H4_1_4_03_FEIL_PR2 5105.05 BOOL  ; HOVEDTAVLE 4.1_SEKSJON_SKUFF        UTLOEST MOTORV. ELLER SIKRING
H4_1_4_03_OK 1604.08 BOOL  ; HOVEDTAVLE 4.1_SEKSJON_SKUFF       DRIFT OG OK
H4_1_4_03_OK_PR2 5105.04 BOOL  ; HOVEDTAVLE 4.1_SEKSJON_SKUFF       DRIFT OG OK
H4_1_4_04_AUTO 1604.09 BOOL  ; HOVEDTAVLE 4.1_SEKSJON_SKUFF        DRIFTSIGN. FRA  NODE1_4
H4_1_4_04_AUTO_PR2 5003.03 BOOL  ; HOVEDTAVLE 4.1_SEKSJON_SKUFF        DRIFTSIGN. FRA  NODE1_4
H4_1_4_04_FEIL 1604.10 BOOL  ; HOVEDTAVLE 4.1_SEKSJON_SKUFF        UTLOEST MOTORV. ELLER SIKRING
H4_1_4_04_FEIL_PR2 5105.07 BOOL  ; HOVEDTAVLE 4.1_SEKSJON_SKUFF        UTLOEST MOTORV. ELLER SIKRING
H4_1_4_04_OK 1604.11 BOOL  ; HOVEDTAVLE 4.1_SEKSJON_SKUFF       DRIFT OG OK
H4_1_4_04_OK_PR2 5105.06 BOOL  ; HOVEDTAVLE 4.1_SEKSJON_SKUFF       DRIFT OG OK
H4_1_4_05_AUTO 1604.12 BOOL  ; HOVEDTAVLE 4.1_SEKSJON_SKUFF        DRIFTSIGN. FRA  NODE1_4
H4_1_4_05_AUTO_PR2 5003.04 BOOL  ; HOVEDTAVLE 4.1_SEKSJON_SKUFF        DRIFTSIGN. FRA  NODE1_4
H4_1_4_05_FEIL 1604.13 BOOL  ; HOVEDTAVLE 4.1_SEKSJON_SKUFF        UTLOEST MOTORV. ELLER SIKRING
H4_1_4_05_FEIL_PR2 5106.01 BOOL  ; HOVEDTAVLE 4.1_SEKSJON_SKUFF        UTLOEST MOTORV. ELLER SIKRING
H4_1_4_05_OK 1604.14 BOOL  ; HOVEDTAVLE 4.1_SEKSJON_SKUFF       DRIFT OG OK
H4_1_4_05_OK_PR2 5106.00 BOOL  ; HOVEDTAVLE 4.1_SEKSJON_SKUFF       DRIFT OG OK
H4_1_4_06_AUTO 1605.00 BOOL  ; HOVEDTAVLE 4.1_SEKSJON_SKUFF        DRIFTSIGN. FRA  NODE1_4
H4_1_4_06_AUTO_PR2 5003.05 BOOL  ; HOVEDTAVLE 4.1_SEKSJON_SKUFF        DRIFTSIGN. FRA  NODE1_4
H4_1_4_06_FEIL 1605.01 BOOL  ; HOVEDTAVLE 4.1_SEKSJON_SKUFF        UTLOEST MOTORV. ELLER SIKRING
H4_1_4_06_FEIL_PR2 5106.03 BOOL  ; HOVEDTAVLE 4.1_SEKSJON_SKUFF        UTLOEST MOTORV. ELLER SIKRING
H4_1_4_06_OK 1605.02 BOOL  ; HOVEDTAVLE 4.1_SEKSJON_SKUFF       DRIFT OG OK
H4_1_4_06_OK_PR2 5106.02 BOOL  ; HOVEDTAVLE 4.1_SEKSJON_SKUFF       DRIFT OG OK
H4_1_4_07_AUTO 1605.03 BOOL  ; HOVEDTAVLE 4.1_SEKSJON_SKUFF        DRIFTSIGN. FRA  NODE1_4
H4_1_4_07_AUTO_PR2 5003.06 BOOL  ; HOVEDTAVLE 4.1_SEKSJON_SKUFF        DRIFTSIGN. FRA  NODE1_4
H4_1_4_07_FEIL 1605.04 BOOL  ; HOVEDTAVLE 4.1_SEKSJON_SKUFF        UTLOEST MOTORV. ELLER SIKRING
H4_1_4_07_FEIL_PR2 5106.05 BOOL  ; HOVEDTAVLE 4.1_SEKSJON_SKUFF        UTLOEST MOTORV. ELLER SIKRING
H4_1_4_07_OK 1605.05 BOOL  ; HOVEDTAVLE 4.1_SEKSJON_SKUFF       DRIFT OG OK
H4_1_4_07_OK_PR2 5106.04 BOOL  ; HOVEDTAVLE 4.1_SEKSJON_SKUFF       DRIFT OG OK
H4_1_4_08_AUTO 1605.06 BOOL  ; HOVEDTAVLE 4.1_SEKSJON_SKUFF        DRIFTSIGN. FRA  NODE1_4
H4_1_4_08_AUTO_PR2 5003.07 BOOL  ; HOVEDTAVLE 4.1_SEKSJON_SKUFF        DRIFTSIGN. FRA  NODE1_4
H4_1_4_08_FEIL 1605.07 BOOL  ; HOVEDTAVLE 4.1_SEKSJON_SKUFF        UTLOEST MOTORV. ELLER SIKRING
H4_1_4_08_FEIL_PR2 5106.07 BOOL  ; HOVEDTAVLE 4.1_SEKSJON_SKUFF        UTLOEST MOTORV. ELLER SIKRING
H4_1_4_08_OK 1605.08 BOOL  ; HOVEDTAVLE 4.1_SEKSJON_SKUFF       DRIFT OG OK
H4_1_4_08_OK_PR2 5106.06 BOOL  ; HOVEDTAVLE 4.1_SEKSJON_SKUFF       DRIFT OG OK
H4_1_4_09_AUTO 1605.09 BOOL  ; HOVEDTAVLE 4.1_SEKSJON_SKUFF        DRIFTSIGN. FRA  NODE1_4
H4_1_4_09_AUTO_PR2 5004.00 BOOL  ; HOVEDTAVLE 4.1_SEKSJON_SKUFF        DRIFTSIGN. FRA  NODE1_4
H4_1_4_09_FEIL 1605.10 BOOL  ; HOVEDTAVLE 4.1_SEKSJON_SKUFF        UTLOEST MOTORV. ELLER SIKRING
H4_1_4_09_FEIL_PR2 5107.01 BOOL  ; HOVEDTAVLE 4.1_SEKSJON_SKUFF        UTLOEST MOTORV. ELLER SIKRING
H4_1_4_09_OK 1605.11 BOOL  ; HOVEDTAVLE 4.1_SEKSJON_SKUFF       DRIFT OG OK
H4_1_4_09_OK_PR2 5107.00 BOOL  ; HOVEDTAVLE 4.1_SEKSJON_SKUFF       DRIFT OG OK
H4_1_4_10_AUTO 1605.12 BOOL  ; HOVEDTAVLE 4.1_SEKSJON_SKUFF        DRIFTSIGN. FRA  NODE1_4
H4_1_4_10_AUTO_PR2 5004.01 BOOL  ; HOVEDTAVLE 4.1_SEKSJON_SKUFF        DRIFTSIGN. FRA  NODE1_4
H4_1_4_10_FEIL 1605.13 BOOL  ; HOVEDTAVLE 4.1_SEKSJON_SKUFF        UTLOEST MOTORV. ELLER SIKRING
H4_1_4_10_FEIL_PR2 5107.03 BOOL  ; HOVEDTAVLE 4.1_SEKSJON_SKUFF        UTLOEST MOTORV. ELLER SIKRING
H4_1_4_10_OK 1605.14 BOOL  ; HOVEDTAVLE 4.1_SEKSJON_SKUFF       DRIFT OG OK
H4_1_4_10_OK_PR2 5107.02 BOOL  ; HOVEDTAVLE 4.1_SEKSJON_SKUFF       DRIFT OG OK
H4_1_5_01_AUTO 1606.00 BOOL  ; HOVEDTAVLE 4.1_SEKSJON_SKUFF        DRIFTSIGN. FRA  NODE1_4
H4_1_5_01_AUTO_PR2 5005.00 BOOL  ; HOVEDTAVLE 4.1_SEKSJON_SKUFF        DRIFTSIGN. FRA  NODE1_4
H4_1_5_01_FEIL 1606.01 BOOL  ; HOVEDTAVLE 4.1_SEKSJON_SKUFF        UTLOEST MOTORV. ELLER SIKRING
H4_1_5_01_FEIL_PR2 5108.01 BOOL  ; HOVEDTAVLE 4.1_SEKSJON_SKUFF        UTLOEST MOTORV. ELLER SIKRING
H4_1_5_01_OK 1606.02 BOOL  ; HOVEDTAVLE 4.1_SEKSJON_SKUFF       DRIFT OG OK
H4_1_5_01_OK_PR2 5108.00 BOOL  ; HOVEDTAVLE 4.1_SEKSJON_SKUFF       DRIFT OG OK
H4_1_5_02_AUTO 1606.03 BOOL  ; HOVEDTAVLE 4.1_SEKSJON_SKUFF        DRIFTSIGN. FRA  NODE1_4
H4_1_5_02_AUTO_PR2 5005.01 BOOL  ; HOVEDTAVLE 4.1_SEKSJON_SKUFF        DRIFTSIGN. FRA  NODE1_4
H4_1_5_02_FEIL 1606.04 BOOL  ; HOVEDTAVLE 4.1_SEKSJON_SKUFF        UTLOEST MOTORV. ELLER SIKRING
H4_1_5_02_FEIL_PR2 5108.03 BOOL  ; HOVEDTAVLE 4.1_SEKSJON_SKUFF        UTLOEST MOTORV. ELLER SIKRING
H4_1_5_02_OK 1606.05 BOOL  ; HOVEDTAVLE 4.1_SEKSJON_SKUFF       DRIFT OG OK
H4_1_5_02_OK_PR2 5108.02 BOOL  ; HOVEDTAVLE 4.1_SEKSJON_SKUFF       DRIFT OG OK
H4_1_5_03_AUTO 1606.06 BOOL  ; HOVEDTAVLE 4.1_SEKSJON_SKUFF        DRIFTSIGN. FRA  NODE1_4
H4_1_5_03_AUTO_PR2 5005.02 BOOL  ; HOVEDTAVLE 4.1_SEKSJON_SKUFF        DRIFTSIGN. FRA  NODE1_4
H4_1_5_03_FEIL 1606.07 BOOL  ; HOVEDTAVLE 4.1_SEKSJON_SKUFF        UTLOEST MOTORV. ELLER SIKRING
H4_1_5_03_FEIL_PR2 5108.05 BOOL  ; HOVEDTAVLE 4.1_SEKSJON_SKUFF        UTLOEST MOTORV. ELLER SIKRING
H4_1_5_03_OK 1606.08 BOOL  ; HOVEDTAVLE 4.1_SEKSJON_SKUFF       DRIFT OG OK
H4_1_5_03_OK_PR2 5108.04 BOOL  ; HOVEDTAVLE 4.1_SEKSJON_SKUFF       DRIFT OG OK
H4_1_5_04_AUTO 1606.09 BOOL  ; HOVEDTAVLE 4.1_SEKSJON_SKUFF        DRIFTSIGN. FRA  NODE1_4
H4_1_5_04_AUTO_PR2 5005.03 BOOL  ; HOVEDTAVLE 4.1_SEKSJON_SKUFF        DRIFTSIGN. FRA  NODE1_4
H4_1_5_04_FEIL 1606.10 BOOL  ; HOVEDTAVLE 4.1_SEKSJON_SKUFF        UTLOEST MOTORV. ELLER SIKRING
H4_1_5_04_FEIL_PR2 5108.07 BOOL  ; HOVEDTAVLE 4.1_SEKSJON_SKUFF        UTLOEST MOTORV. ELLER SIKRING
H4_1_5_04_OK 1606.11 BOOL  ; HOVEDTAVLE 4.1_SEKSJON_SKUFF       DRIFT OG OK
H4_1_5_04_OK_PR2 5108.06 BOOL  ; HOVEDTAVLE 4.1_SEKSJON_SKUFF       DRIFT OG OK
H4_1_5_05_AUTO 1606.12 BOOL  ; HOVEDTAVLE 4.1_SEKSJON_SKUFF        DRIFTSIGN. FRA  NODE1_4
H4_1_5_05_AUTO_PR2 5005.04 BOOL  ; HOVEDTAVLE 4.1_SEKSJON_SKUFF        DRIFTSIGN. FRA  NODE1_4
H4_1_5_05_FEIL 1606.13 BOOL  ; HOVEDTAVLE 4.1_SEKSJON_SKUFF        UTLOEST MOTORV. ELLER SIKRING
H4_1_5_05_FEIL_PR2 5109.01 BOOL  ; HOVEDTAVLE 4.1_SEKSJON_SKUFF        UTLOEST MOTORV. ELLER SIKRING
H4_1_5_05_OK 1606.14 BOOL  ; HOVEDTAVLE 4.1_SEKSJON_SKUFF       DRIFT OG OK
H4_1_5_05_OK_PR2 5109.00 BOOL  ; HOVEDTAVLE 4.1_SEKSJON_SKUFF       DRIFT OG OK
H4_1_5_06_AUTO 1607.00 BOOL  ; HOVEDTAVLE 4.1_SEKSJON_SKUFF        DRIFTSIGN. FRA  NODE1_4
H4_1_5_06_AUTO_PR2 5005.05 BOOL  ; HOVEDTAVLE 4.1_SEKSJON_SKUFF        DRIFTSIGN. FRA  NODE1_4
H4_1_5_06_FEIL 1607.01 BOOL  ; HOVEDTAVLE 4.1_SEKSJON_SKUFF        UTLOEST MOTORV. ELLER SIKRING
H4_1_5_06_FEIL_PR2 5109.03 BOOL  ; HOVEDTAVLE 4.1_SEKSJON_SKUFF        UTLOEST MOTORV. ELLER SIKRING
H4_1_5_06_OK 1607.02 BOOL  ; HOVEDTAVLE 4.1_SEKSJON_SKUFF       DRIFT OG OK
H4_1_5_06_OK_PR2 5109.02 BOOL  ; HOVEDTAVLE 4.1_SEKSJON_SKUFF       DRIFT OG OK
H4_1_6_01_AUTO 1608.00 BOOL  ; HOVEDTAVLE 4.1_SEKSJON_SKUFF        DRIFTSIGN. FRA  NODE1_4
H4_1_6_01_AUTO_PR2 5006.00 BOOL  ; HOVEDTAVLE 4.1_SEKSJON_SKUFF        DRIFTSIGN. FRA  NODE1_4
H4_1_6_01_FEIL 1608.01 BOOL  ; HOVEDTAVLE 4.1_SEKSJON_SKUFF        UTLOEST MOTORV. ELLER SIKRING
H4_1_6_01_FEIL_PR2 5110.01 BOOL  ; HOVEDTAVLE 4.1_SEKSJON_SKUFF        UTLOEST MOTORV. ELLER SIKRING
H4_1_6_01_OK 1608.02 BOOL  ; HOVEDTAVLE 4.1_SEKSJON_SKUFF       DRIFT OG OK
H4_1_6_01_OK_PR2 5110.00 BOOL  ; HOVEDTAVLE 4.1_SEKSJON_SKUFF       DRIFT OG OK
H4_1_6_02_AUTO 1608.03 BOOL  ; HOVEDTAVLE 4.1_SEKSJON_SKUFF        DRIFTSIGN. FRA  NODE1_4
H4_1_6_02_AUTO_PR2 5006.01 BOOL  ; HOVEDTAVLE 4.1_SEKSJON_SKUFF        DRIFTSIGN. FRA  NODE1_4
H4_1_6_02_FEIL 1608.04 BOOL  ; HOVEDTAVLE 4.1_SEKSJON_SKUFF        UTLOEST MOTORV. ELLER SIKRING
H4_1_6_02_FEIL_PR2 5110.03 BOOL  ; HOVEDTAVLE 4.1_SEKSJON_SKUFF        UTLOEST MOTORV. ELLER SIKRING
H4_1_6_02_OK 1608.05 BOOL  ; HOVEDTAVLE 4.1_SEKSJON_SKUFF       DRIFT OG OK
H4_1_6_02_OK_PR2 5110.02 BOOL  ; HOVEDTAVLE 4.1_SEKSJON_SKUFF       DRIFT OG OK
H4_1_6_03_AUTO 1608.06 BOOL  ; HOVEDTAVLE 4.1_SEKSJON_SKUFF        DRIFTSIGN. FRA  NODE1_4
H4_1_6_03_AUTO_PR2 5006.02 BOOL  ; HOVEDTAVLE 4.1_SEKSJON_SKUFF        DRIFTSIGN. FRA  NODE1_4
H4_1_6_03_FEIL 1608.07 BOOL  ; HOVEDTAVLE 4.1_SEKSJON_SKUFF        UTLOEST MOTORV. ELLER SIKRING
H4_1_6_03_FEIL_PR2 5110.05 BOOL  ; HOVEDTAVLE 4.1_SEKSJON_SKUFF        UTLOEST MOTORV. ELLER SIKRING
H4_1_6_03_OK 1608.08 BOOL  ; HOVEDTAVLE 4.1_SEKSJON_SKUFF       DRIFT OG OK
H4_1_6_03_OK_PR2 5110.04 BOOL  ; HOVEDTAVLE 4.1_SEKSJON_SKUFF       DRIFT OG OK
H4_1_6_04_AUTO 1608.09 BOOL  ; HOVEDTAVLE 4.1_SEKSJON_SKUFF        DRIFTSIGN. FRA  NODE1_4
H4_1_6_04_AUTO_PR2 5006.03 BOOL  ; HOVEDTAVLE 4.1_SEKSJON_SKUFF        DRIFTSIGN. FRA  NODE1_4
H4_1_6_04_FEIL 1608.10 BOOL  ; HOVEDTAVLE 4.1_SEKSJON_SKUFF        UTLOEST MOTORV. ELLER SIKRING
H4_1_6_04_FEIL_PR2 5110.07 BOOL  ; HOVEDTAVLE 4.1_SEKSJON_SKUFF        UTLOEST MOTORV. ELLER SIKRING
H4_1_6_04_OK 1608.11 BOOL  ; HOVEDTAVLE 4.1_SEKSJON_SKUFF       DRIFT OG OK
H4_1_6_04_OK_PR2 5110.06 BOOL  ; HOVEDTAVLE 4.1_SEKSJON_SKUFF       DRIFT OG OK
H4_1_6_05_AUTO 1608.12 BOOL  ; HOVEDTAVLE 4.1_SEKSJON_SKUFF        DRIFTSIGN. FRA  NODE1_4
H4_1_6_05_AUTO_PR2 5006.04 BOOL  ; HOVEDTAVLE 4.1_SEKSJON_SKUFF        DRIFTSIGN. FRA  NODE1_4
H4_1_6_05_FEIL 1608.13 BOOL  ; HOVEDTAVLE 4.1_SEKSJON_SKUFF        UTLOEST MOTORV. ELLER SIKRING
H4_1_6_05_FEIL_PR2 5111.01 BOOL  ; HOVEDTAVLE 4.1_SEKSJON_SKUFF        UTLOEST MOTORV. ELLER SIKRING
H4_1_6_05_OK 1608.14 BOOL  ; HOVEDTAVLE 4.1_SEKSJON_SKUFF       DRIFT OG OK
H4_1_6_05_OK_PR2 5111.00 BOOL  ; HOVEDTAVLE 4.1_SEKSJON_SKUFF       DRIFT OG OK
H4_1_6_06_AUTO 1609.00 BOOL  ; HOVEDTAVLE 4.1_SEKSJON_SKUFF        DRIFTSIGN. FRA  NODE1_4
H4_1_6_06_AUTO_PR2 5006.05 BOOL  ; HOVEDTAVLE 4.1_SEKSJON_SKUFF        DRIFTSIGN. FRA  NODE1_4
H4_1_6_06_FEIL 1609.01 BOOL  ; HOVEDTAVLE 4.1_SEKSJON_SKUFF        UTLOEST MOTORV. ELLER SIKRING
H4_1_6_06_FEIL_PR2 5111.03 BOOL  ; HOVEDTAVLE 4.1_SEKSJON_SKUFF        UTLOEST MOTORV. ELLER SIKRING
H4_1_6_06_OK 1609.02 BOOL  ; HOVEDTAVLE 4.1_SEKSJON_SKUFF       DRIFT OG OK
H4_1_6_06_OK_PR2 5111.02 BOOL  ; HOVEDTAVLE 4.1_SEKSJON_SKUFF       DRIFT OG OK
H4_1_6_07_AUTO 1609.03 BOOL  ; HOVEDTAVLE 4.1_SEKSJON_SKUFF        DRIFTSIGN. FRA  NODE1_4
H4_1_6_07_AUTO_PR2 5006.06 BOOL  ; HOVEDTAVLE 4.1_SEKSJON_SKUFF        DRIFTSIGN. FRA  NODE1_4
H4_1_6_07_FEIL 1609.04 BOOL  ; HOVEDTAVLE 4.1_SEKSJON_SKUFF        UTLOEST MOTORV. ELLER SIKRING
H4_1_6_07_FEIL_PR2 5111.05 BOOL  ; HOVEDTAVLE 4.1_SEKSJON_SKUFF        UTLOEST MOTORV. ELLER SIKRING
H4_1_6_07_OK 1609.05 BOOL  ; HOVEDTAVLE 4.1_SEKSJON_SKUFF       DRIFT OG OK
H4_1_6_07_OK_PR2 5111.04 BOOL  ; HOVEDTAVLE 4.1_SEKSJON_SKUFF       DRIFT OG OK
H4_1_6_08_AUTO 1609.06 BOOL  ; HOVEDTAVLE 4.1_SEKSJON_SKUFF        DRIFTSIGN. FRA  NODE1_4
H4_1_6_08_AUTO_PR2 5006.07 BOOL  ; HOVEDTAVLE 4.1_SEKSJON_SKUFF        DRIFTSIGN. FRA  NODE1_4
H4_1_6_08_FEIL 1609.07 BOOL  ; HOVEDTAVLE 4.1_SEKSJON_SKUFF        UTLOEST MOTORV. ELLER SIKRING
H4_1_6_08_FEIL_PR2 5111.07 BOOL  ; HOVEDTAVLE 4.1_SEKSJON_SKUFF        UTLOEST MOTORV. ELLER SIKRING
H4_1_6_08_OK 1609.08 BOOL  ; HOVEDTAVLE 4.1_SEKSJON_SKUFF       DRIFT OG OK
H4_1_6_08_OK_PR2 5111.06 BOOL  ; HOVEDTAVLE 4.1_SEKSJON_SKUFF       DRIFT OG OK
H4_1_6_09_AUTO 1609.09 BOOL  ; HOVEDTAVLE 4.1_SEKSJON_SKUFF        DRIFTSIGN. FRA  NODE1_4
H4_1_6_09_AUTO_PR2 5007.00 BOOL  ; HOVEDTAVLE 4.1_SEKSJON_SKUFF        DRIFTSIGN. FRA  NODE1_4
H4_1_6_09_FEIL 1609.10 BOOL  ; HOVEDTAVLE 4.1_SEKSJON_SKUFF        UTLOEST MOTORV. ELLER SIKRING
H4_1_6_09_FEIL_PR2 5112.01 BOOL  ; HOVEDTAVLE 4.1_SEKSJON_SKUFF        UTLOEST MOTORV. ELLER SIKRING
H4_1_6_09_OK 1609.11 BOOL  ; HOVEDTAVLE 4.1_SEKSJON_SKUFF       DRIFT OG OK
H4_1_6_09_OK_PR2 5112.00 BOOL  ; HOVEDTAVLE 4.1_SEKSJON_SKUFF       DRIFT OG OK
H4_1_6_10_AUTO 1609.12 BOOL  ; HOVEDTAVLE 4.1_SEKSJON_SKUFF        DRIFTSIGN. FRA  NODE1_4
H4_1_6_10_AUTO_PR2 5007.01 BOOL  ; HOVEDTAVLE 4.1_SEKSJON_SKUFF        DRIFTSIGN. FRA  NODE1_4
H4_1_6_10_FEIL 1609.13 BOOL  ; HOVEDTAVLE 4.1_SEKSJON_SKUFF        UTLOEST MOTORV. ELLER SIKRING
H4_1_6_10_OK 1609.14 BOOL  ; HOVEDTAVLE 4.1_SEKSJON_SKUFF       DRIFT OG OK
H4_1_6_10_OK_PR2 5112.02 BOOL  ; HOVEDTAVLE 4.1_SEKSJON_SKUFF       DRIFT OG OK
HAST_UT_P8002 D20148 INT
HAST_UT_P8003 D20248 INT
HAST_UT_P8010 D20048 INT
HENGER01_0_STATUS 521.01 BOOL  ; XN4_BIL1_. Alle objekter som ikke betjenes er ok
HENGER01_1_STATUS 521.02 BOOL  ; XN4_BIL1_. Alle utstyrte objekter i 1.fase er ok
HENGER01_2_STAT 521.03 BOOL  ; X Alle utstyrte objekter er ok. Pgm = ok.
HENGER01_DRIFT 521.00 BOOL  ; XN4_BIL1_ i drift
HENGER01_FEIL 521.04 BOOL  ; XFeil
HENGER01_FEILTID 521.05 BOOL  ; X
HENGER01_HJ0 421.04 BOOL  ; X
HENGER01_HJ1 421.05 BOOL  ; X
HENGER01_INDIVID_INNE 521.15 BOOL  ; XIndividadresse er
HENGER01_INDKON 521.06 BOOL  ; XKontr. at bare en individadresse er hoey.
HENGER01_KOEINLES D5218 CHANNEL  ; XINNLESNING AVKOMMANDOVERDIER FRA D3000
HENGER01_KOELES 321.14 BOOL  ; SPERR INNLESNING TIL KOE-REGISTER.
HENGER01_KOEPLASS_1 D5210 CHANNEL  ; XFOERST I KOE
HENGER01_KOEPLASS_2 D5212 CHANNEL  ; X
HENGER01_KOEPLASS_3 D5214 CHANNEL  ; X
HENGER01_KOEPLASS_4 D5216 CHANNEL  ; X
HENGER01_KOMMANDO_KOE 321.15 BOOL  ; D3000 VERDI KAN OVERFOERES TIL KOE-REGISTER.
HENGER01_OFF_IMP 521.14 BOOL  ; X
HENGER01_ONIMPULS 521.11 BOOL  ; XN4_BIL1_Startimpuls for  program
HENGER01_RESET 521.09 BOOL  ; XN4_BIL1. Stopp og nedkobling av programmet
HENGER01_START 521.07 BOOL  ; Xprogram starter
HENGER01_STARTIMPULS 521.10 BOOL  ; XN4_BIL1. Startimpuls.
HENGER01_T03_IND 1221.00 BOOL  ; X
HENGER01_T04_IND 1221.01 BOOL
HENGER01_T05_IND 1221.02 BOOL  ; X
HENGER01_TID_S T0521 BOOL  ; X
HENGER01_TID_T 521 NUMBER
HENGER01_TIL_T03_VALG 321.00 BOOL  ; NDIVIDVALG FRA KOEREGISTER.
HENGER01_TIL_T04_VALG 321.01 BOOL  ; INDIVIDVALG FRA KOEREGISTER.
HENGER01_TIL_T05_VALG 321.02 BOOL  ; INDIVIDVALG FRA KOEREGISTER.
HENGER02_0_STATUS 523.01 BOOL  ; XN4_BIL1_. Alle objekter som ikke betjenes er ok
HENGER02_1_STATUS 523.02 BOOL  ; XN4_BIL1_. Alle utstyrte objekter i 1.fase er ok
HENGER02_2_STAT 523.03 BOOL  ; X Alle utstyrte objekter er ok. Pgm = ok.
HENGER02_DRIFT 523.00 BOOL  ; XN4_BIL1_ i drift
HENGER02_FEIL 523.04 BOOL  ; XFeil
HENGER02_FEILTID 523.05 BOOL  ; X
HENGER02_HJ0 423.04 BOOL  ; X
HENGER02_HJ1 423.05 BOOL  ; X
HENGER02_INDIVID_INNE 523.15 BOOL  ; XIndividadresse er
HENGER02_INDKON 523.06 BOOL  ; XKontr. at bare en individadresse er hoey.
HENGER02_KOELES 323.14 BOOL  ; SPERR INNLESNING TIL KOE-REGISTER.
HENGER02_KOEPLASS_1 D5230 CHANNEL  ; XFOERST I KOE
HENGER02_KOEPLASS_2 D5232 CHANNEL  ; X
HENGER02_KOEPLASS_3 D5234 CHANNEL  ; X
HENGER02_KOMMANDO_KOE 323.15 BOOL  ; D3000 VERDI KAN OVERFOERES TIL KOE-REGISTER.
HENGER02_OFF_IMP 523.14 BOOL  ; X
HENGER02_ONIMPULS 523.11 BOOL  ; XN4_BIL1_Startimpuls for  program
HENGER02_RESET 523.09 BOOL  ; XN4_BIL1. Stopp og nedkobling av programmet
HENGER02_START 523.07 BOOL  ; Xprogram starter
HENGER02_STARTIMPULS 523.10 BOOL  ; XN4_BIL1. Startimpuls.
HENGER02_T03_IND 1223.00 BOOL  ; X
HENGER02_T04_IND 1223.01 BOOL  ; XN4_BIL1_TIL_T04_INDIVID
HENGER02_T05_IND 1223.02 BOOL  ; X
HENGER02_TID_S T0523 BOOL  ; X
HENGER02_TID_T 523 NUMBER
HENGER02_TIL_T03_VALG 323.00 BOOL  ; INDIVIDVALG FRA KOEREGISTER.
HENGER02_TIL_T04 323.01 BOOL  ; INDIVIDVALG FRA KOEREGISTER.
HENGER02_TIL_T05_VALG 323.02 BOOL  ; INDIVIDVALG FRA KOEREGISTER.
HENGER02_TMU_USIKRET 1223.15 BOOL  ; XN4_BIL1_USIKRET
HENSTANDSFLOETE 4520.06 BOOL
HIGH_LEVEL_BLK21 HIGH_LEVEL
HIGH_LEVEL_BLK22 HIGH_LEVEL
HIGH_LEVEL_BLK23 HIGH_LEVEL
HJ133700 942.00 BOOL
HJ133709 942.01 BOOL
HJ1_C12_33_36 933.00 BOOL
HJ1_C13_34_37 933.02 BOOL
HJ1_C14_35_38 933.04 BOOL
HJ1_C15 933.06 BOOL
HJ1_KLAPR 942.13 BOOL
HJ1_V8223_AUT 942.15 BOOL
HJ1_V8224 943.00 BOOL
HJ1_V8323 943.01 BOOL
HJ1_V8324 943.02 BOOL
HJ1_VANNFYLL_T84 994.00 BOOL
HJ2_C12_33_36 933.01 BOOL
HJ2_C13_34_37 933.03 BOOL
HJ2_C14_35_38 933.05 BOOL
HJ2_K4_LUT_SYRE_CALL 942.03 BOOL  ; ADRESSE =1= PASTEUR OENSKER LUT ELLER SYRE
HJ2_KLAPR 942.14 BOOL
HJ2_V4302 960.11 BOOL
HJ2_V8221 942.07 BOOL
HJ2_V8321 942.10 BOOL
HJ3_V8221 942.08 BOOL
HJ3_V8321 942.11 BOOL
HJ4_V8221 942.09 BOOL
HJ4_V8231 942.12 BOOL
HJP8004_4 942.04 BOOL
HJ_BLAAS_LAB 960.08 BOOL
HJ_BLAAS_UHT 960.09 BOOL
HJ_NULLST_Q8001 902.14 BOOL
HJ_NULLST_Q8002 912.14 BOOL
HJ_NULLST_Q8003 922.14 BOOL
HJ_OPPSAML_OK 960.14 BOOL
HJ_SLANGE_UHT 960.04 BOOL
HJ_SPJ_LAB 960.02 BOOL
HJ_SPJ_UHT 960.03 BOOL
HJ_V8214 942.05 BOOL
HJ_V8314 942.06 BOOL
HJ_VACUUM 960.00 BOOL
HJ_VANN 994.01 BOOL
HJ_VANNF_PASVASK 943.03 BOOL  ; VASK_PASTEURER_I_DRIFT
HJ_V_4302_UT 960.10 BOOL
HL_BLK21 4501.00 BOOL
HL_BLK22 4511.00 BOOL
HL_BLK23 4521.00 BOOL
HL_T03 600.00 BOOL
HL_T03_FORSINKELSE T0610 BOOL  ; TID SOM FORSINKER  TOPPVARSEL PAA T03
HL_T03_PLS1 4600.00 BOOL
HL_T04 602.00 BOOL
HL_T04_FORSINKELSE T0620 BOOL  ; TID SOM FORSINKER  TOPPVARSEL PAA T04
HL_T04_PLS1 4600.02 BOOL
HL_T05 604.00 BOOL
HL_T05_FORSINKELSE T0640 BOOL  ; TID SOM FORSINKER  TOPPVARSEL PAA T05
HL_T05_PLS1 4600.04 BOOL
HL_T24_01 750.00 BOOL
HL_T24_01_FORSINKELSE_S T0668 BOOL  ; TID SOM FORSINKER  TOPPVARSEL PAA T24.01
HL_T24_01_FORSINKELSE_T 0668 NUMBER  ; TID SOM FORSINKER  TOPPVARSEL PAA T24.01
HL_T2701 688.00 BOOL
HL_T2702 689.00 BOOL
HL_T2703 690.00 BOOL
HL_T40 648.00 BOOL
HL_T40_FORSINKELSE_S T0612 BOOL  ; TID SOM FORSINKER  TOPPVARSEL PAA T40
HL_T40_FORSINKELSE_T 0612 NUMBER  ; TID SOM FORSINKER  TOPPVARSEL PAA T40
HL_T41 649.00 BOOL
HL_T41_FORSINKELSE_S T0614 BOOL  ; TID SOM FORSINKER  TOPPVARSEL PAA T41
HL_T41_FORSINKELSE_T 0614 NUMBER  ; TID SOM FORSINKER  TOPPVARSEL PAA T41
HL_T81 1401.10 BOOL
HL_T82 1402.10 BOOL  ; HL- T 82 Luttank.
HL_T83 1403.10 BOOL  ; HL- T 83 Syretank.
HL_T84 1404.10 BOOL  ; HL- T 84 Hetvanntank.
HOLDSIGNAL_TANKVASK_K1 1306.10 BOOL
HOLDSIGNAL_TANKVASK_K2 1316.10 BOOL
HOLDSIGNAL_TANKVASK_K3 1326.10 BOOL
HOMO21_I_LINJE 4500.07 BOOL
HOMO21_TR1_BEREGN D1772 REAL
HOMO21_TR1_FORV D1770 REAL
HOMO22_I_LINJE 4510.07 BOOL
HOMO22_TR1_OPPSKALER OPPSKALERING
HOMO22_TR2_OPPSKALER OPPSKALERING
HOMO_21_SOETMELK_INN 4804.01 BOOL
HOMO_21_SOETMELK_I_HOMO 4804.02 BOOL
HOMO_21_SOETMELK_TIL_HOMO 4804.03 BOOL
HOMO_21_TRYKK1 D1790 CHANNEL
HOMO_21_TRYKK1_PR5 D1794 CHANNEL
HOMO_21_TRYKK2 D1792 CHANNEL
HOMO_21_TRYKK2_PR5 D1796 CHANNEL
HOMO_22_ER_HAST D3752 REAL
HOMO_22_HAST D1804 CHANNEL
HOMO_22_HAST_RAA D1814 CHANNEL
HOMO_22_TRYKK1 D1800 CHANNEL
HOMO_22_TRYKK2 D1802 CHANNEL
HP1_K4_LUT_SYRE_CALL 942.02 BOOL  ; ADRESSE =1= PASTEUR OENSKER LUT ELLER SYRE
HURTIG_BLINK 999.02 BOOL  ; 0,2 SEKUNERS BINK
HYST_K1_GRM D8648 INT
INN_B8402 5115 CHANNEL
INN_V8001_PROFI 5116.00 BOOL
K1_1_VMF_FERDIG 1306.00 BOOL
K1_COND_HJ1 903.05 BOOL
K1_DESINFEKSJON 1304.02 BOOL
K1_FASEFORLENG 1305.15 BOOL  ; FORLENG AKTUEL VASKEFASE/TRINN.
K1_FASEF_OFFIMP 1306.06 BOOL  ; FERDIG-OFF-IMPULS.
K1_FEIL_LINJEPGM 1306.15 BOOL  ; FEIL PAA AKTUELL VASK
K1_FORSINK_FEIL_FLOW T0034 BOOL
K1_FORSINK_SIRK T0160 BOOL
K1_FORSKYLL 1304.05 BOOL
K1_FORSK_LUT 1304.00 BOOL  ; FORSKYLL_LUT
K1_FORSK_LUT_DES 1304.01 BOOL  ; FORSKYLLING- LUT-DESINFEKSJON
K1_GRAFIKKTR_HJ1 901.08 BOOL
K1_GRM_FERDIG 1305.08 BOOL  ; GRENSEMELKFASEN AVSLUTTET.
K1_GRM_HJ1 901.02 BOOL
K1_GRM_RESET 1306.04 BOOL  ; RESET-PULS ETTER GRENSEMELKFASEN.
K1_GR_MELK_I_SYSTEM 1308.00 BOOL
K1_HJ1_TIL_TANK 1308.07 BOOL  ; ETTERRENNING_VED_TANKVASK
K1_HJ2_TIL_TANK_K1 1308.08 BOOL  ; ETTERRENNING_VASK_HENGER
K1_KLAPRING 1306.08 BOOL  ; KLAPRING I FASEN STARTET.
K1_KLAP_SLUTT 1306.09 BOOL  ; KLAPRING I FASEN AVSLUTTET.
K1_KONS_TID_FL 1307.00 BOOL  ; KURS1 KONS. ETTER VENTETID
K1_LUT 1304.04 BOOL  ; LUT
K1_LUTVASK 1306.01 BOOL  ; DET VASKES BARE MED LUT
K1_LUT_DES 1304.03 BOOL  ; LUT OG DESINFEKSJON
K1_LU_ER_STOERRE_PRS 1306.13 BOOL  ; KURS1 LUTKONSENTRASJON I RETUR HOEYERE ENN BOERVERDIEN
K1_NOEDSTOPP 1305.05 BOOL  ; VASKEPROGR. STOPPER OG PUMPENE I VASKEN STOPPER.
K1_SIRKULASJON 1309.00 BOOL
K1_SPERR 1305.07 BOOL
K1_STERT_OK 1305.10 BOOL  ; STERILTEMP. ER OPPNAADD.
K1_SY_ER_STOERRE_PRS 1306.14 BOOL  ; KURS1 SYREKONSENTRASJON I RETUR HOEYERE ENN BOERVERDIEN
K1_TEMP_HJ1 903.06 BOOL
K1_TID_FLOW_BIL_S T0910 BOOL
K1_TID_FLOW_BIL_T 0910 NUMBER
K1_TID_FLOW_HENG_S T0511 BOOL
K1_TID_FLOW_HENG_T 0511 NUMBER
K1_TR01_TID_S C0101 BOOL  ; KURS 1 TRINN 01 TID
K1_TR02_TID_S C0102 BOOL  ; KURS 1 TRINN 02 TID
K1_TR03_TID_PV C103 CHANNEL  ; KURS 1 TRINN 03 TID
K1_TR03_TID_S C0103 BOOL  ; KURS 1 TRINN 03 TID
K1_TR04_TID_S C0104 BOOL  ; KURS 1 TRINN 04 TID
K1_TR05_TID_S C0105 BOOL  ; KURS 1 TRINN 05 TID
K1_TR06_TID_S C0106 BOOL  ; KURS 1 TRINN 06 TID
K1_TR07_TID_PV C107 CHANNEL  ; KURS 1 TRINN 07TID
K1_TR07_TID_S C0107 BOOL  ; KURS 1 TRINN 07TID
K1_TR08_TID_S C0108 BOOL  ; KURS 1 TRINN 08TID
K1_TR09_TID_S C0109 BOOL  ; KURS 1 TRINN 09TID
K1_TR10_TID_S C0110 BOOL  ; KURS 1 TRINN 10-TID
K1_TR11_TID_S C0111 BOOL  ; KURS 1 TRINN 11 TID
K1_TR12_TID_S C0112 BOOL  ; KURS 1 TRINN 12 TID
K1_TR13_TID_S C0113 BOOL  ; KURS 1 TRINN 13 TID
K1_TR14_TID_S C0114 BOOL  ; KURS 1 TRINN 14 TID
K1_TR15_TID_S C0115 BOOL  ; KURS 1 TRINN 15 TID
K1_TR16_TID_S C0116 BOOL  ; KURS 1 TRINN 16 TID
K1_TR17_TID_S C0117 BOOL  ; KURS 1 TRINN 17 TID
K1_TR18_TID_S C0118 BOOL  ; KURS 1 TRINN 18 TID
K1_TR19_TID_S C0119 BOOL  ; KURS 1 TRINN 19 TID
K1_TR20_TID_S C0120 BOOL  ; KURS 1 TRINN 20 TID
K1_TR21_TID_PV C121 CHANNEL  ; KURS 1 TRINN 21 TID
K1_TR21_TID_S C0121 BOOL  ; KURS 1 TRINN 21 TID
K1_TR22_TID_S C0122 BOOL  ; KURS 1 TRINN 22 TID
K1_TR23_TID_S C0123 BOOL  ; KURS 1 TRINN 23 TID
K1_TR24_TID_S C0124 BOOL  ; KURS 1 TRINN 24 TID
K1_TR25_TID_S C0125 BOOL  ; KURS 1 TRINN 25 TID
K1_TR26_TID_S C0126 BOOL  ; KURS 1 TRINN 26 TID
K1_TR27_TID_S C0127 BOOL  ; KURS 1 TRINN 27 TID
K1_TR28_TID_S C0128 BOOL  ; KURS 1 TRINN 28 TID
K1_TR29_TID_S C0129 BOOL  ; KURS 1 TRINN 29 TID
K1_TR30_TID_S C0130 BOOL  ; KURS 1 TRINN 30 TID
K1_TRINNSKIFTE 1307.06 BOOL  ; Trinnskifte i vasken.
K1_TURSTOPP 1305.13 BOOL  ; STANSER TURPUMPENE.
K1_TURTEMP_LAV 1309.01 BOOL
K1_TUR_HJ1 901.03 BOOL
K1_TUR_HJ2 901.04 BOOL
K1_TUR_HJ3 901.05 BOOL
K1_TUR_HJ4 901.06 BOOL
K1_VASK_INNE 1307.05 BOOL
K1_VENT_FOER_LUT 1309.02 BOOL
K1_VENT_TEMPERATUR 1309.03 BOOL
K1_VMFAS_RESET 1306.07 BOOL  ; RESETPULS ETTER AT LUTFASEN ER FERDIG OG SYREFASEN STARTES
K1_VM_KONOK 1305.09 BOOL  ; KONSENTRASJON-VASKEMIDDEL ER OPNAADD I DENNE VASKEFASEN.
K1_V_DRIFT_OK 1300.00 BOOL  ; VASK MELLO TRINN1 OG 30 OG ALT FUNGERER
K1_V_RESET 1306.02 BOOL  ; 0-STILLER VASKEPGM.
K2_1_VMF_FERDIG 1316.00 BOOL
K2_COND_HJ1 913.05 BOOL
K2_DESINFEKSJON 1314.02 BOOL
K2_FASEFORLENG 1315.15 BOOL
K2_FASEF_OFFIMP 1316.06 BOOL  ; FERDIG-OFF-IMPULS.
K2_FEIL_LINJEPGM 1316.15 BOOL
K2_FORSINK_FEIL_FLOW T0134 BOOL
K2_FORSINK_SIRK T0170 BOOL
K2_FORSKYLL 1314.05 BOOL
K2_FORSK_LUT 1314.00 BOOL  ; FORSKYLL_LUT
K2_FORSK_LUT_DES 1314.01 BOOL  ; FORSKYLLING- LUT-DESINFEKSJON
K2_GRAFIKKTR_HJ1 911.08 BOOL
K2_GRM_FERDIG 1315.08 BOOL  ; GRENSEMELKFASEN AVSLUTTET.
K2_GRM_RESET 1316.04 BOOL
K2_GR_MELK_I_SYSTEM 1318.00 BOOL
K2_HJ1_TIL_TANK 1318.07 BOOL  ; ETTERRENNING_VED_TANKVASK
K2_HJ2_TIL_TANK_K2 1318.08 BOOL  ; ETTERRENNING_VED_VASK_HENGER
K2_KLAPRING 1316.08 BOOL
K2_KLAP_SLUTT 1316.09 BOOL  ; KLAPRING I FASEN AVSLUTTET.
K2_KONS_TID_FL 1317.00 BOOL
K2_LUT 1314.04 BOOL  ; LUT
K2_LUTVASK 1316.01 BOOL
K2_LUT_DES 1314.03 BOOL  ; LUT OG DESINFEKSJON
K2_LU_ER_STOERRE_PRS 1316.13 BOOL
K2_NOEDSTOPP 1315.05 BOOL  ; VASKEPROGR. STOPPER OG PUMPENE I VASKEN STOPPER.
K2_SPERR 1315.07 BOOL
K2_STERT_OK 1315.10 BOOL  ; STERILTEMP. ER OPPNAADD
K2_SY_ER_STOERRE_PRS 1316.14 BOOL
K2_TEMP_HJ1 913.06 BOOL
K2_TID_FLOW_BIL_S T0512 BOOL
K2_TID_FLOW_BIL_T 0512 NUMBER
K2_TID_FLOW_HENG_S T0513 BOOL
K2_TID_FLOW_HENG_T 0513 NUMBER
K2_TR01_TID_S C0201 BOOL  ; KURS 2 TRINN 01 TID
K2_TR02_TID_S C0202 BOOL  ; KURS 2 TRINN 2 TID
K2_TR03_TID_PV C203 CHANNEL
K2_TR03_TID_S C0203 BOOL  ; KURS 2 TRINN 03 TID
K2_TR04_TID_S C0204 BOOL  ; KURS 2  TRINN 04 TID
K2_TR05_TID_S C0205 BOOL  ; KURS 2 TRINN 05 TID
K2_TR06_TID_S C0206 BOOL  ; KURS 2 TRINN 06 TID
K2_TR07_TID_PV C207 CHANNEL
K2_TR07_TID_S C0207 BOOL  ; KURS 2 TRINN 07 TID
K2_TR08_TID_S C0208 BOOL  ; KURS 2 TRINN 08 TID
K2_TR09_TID_S C0209 BOOL
K2_TR10_TID_S C0210 BOOL
K2_TR11_TID_S C0211 BOOL  ; KURS 2 TRINN 11 TID
K2_TR12_TID_S C0212 BOOL  ; KURS 2 TRINN 12 TID
K2_TR13_TID_S C0213 BOOL  ; KURS 2 TRINN 13 TID
K2_TR14_TID_S C0214 BOOL
K2_TR15_TID_S C0215 BOOL  ; KURS 2 TRINN 15 TID
K2_TR16_TID_S C0216 BOOL  ; KURS 2 TRINN 16 TID
K2_TR17_TID_S C0217 BOOL  ; KURS 2 TRINN 17 TID
K2_TR18_TID_S C0218 BOOL  ; KURS 2 TRINN18 TID
K2_TR19_TID_S C0219 BOOL  ; KURS 2 TRINN19 TID
K2_TR20_TID_S C0220 BOOL  ; KURS 2 TRINN 20 TID
K2_TR21_TID_PV C221 CHANNEL
K2_TR21_TID_S C0221 BOOL  ; KURS 2 TRINN 21 TID
K2_TR22_TID_S C0222 BOOL  ; KURS 2 TRINN 22
K2_TR23_TID_S C0223 BOOL  ; KURS 2 TRINN 23 TID
K2_TR24_TID_S C0224 BOOL  ; KURS 2 TRINN 24 TID
K2_TR25_TID_S C0225 BOOL  ; KURS 2 TRINN 25 TID
K2_TR26_TID_S C0226 BOOL  ; KURS 2 TRINN 26 TID
K2_TR27_TID_S C0227 BOOL  ; KURS 2 TRINN 27 TID
K2_TR28_TID_S C0228 BOOL  ; KURS 2 TRINN 29 TID
K2_TR29_TID_S C0229 BOOL  ; KURS 2 TRINN 29 TID
K2_TR30_TID_S C0230 BOOL  ; KURS 2 TRINN 30 TID
K2_TRINNSKIFTE 1317.06 BOOL
K2_TURSTOPP 1315.13 BOOL  ; STANSER TURPUMPENE.
K2_TURTEMP_LAV 1319.01 BOOL
K2_TUR_HJ1 911.03 BOOL
K2_TUR_HJ2 911.04 BOOL
K2_TUR_HJ3 911.05 BOOL
K2_TUR_HJ4 911.06 BOOL
K2_VASK_INNE 1317.05 BOOL
K2_VENT_FOER_LUT 1319.02 BOOL
K2_VENT_TEMPERATUR 1319.03 BOOL
K2_VMFAS_RESET 1316.07 BOOL
K2_VM_KONOK 1315.09 BOOL  ; KONSENTRASJON-VASKEMIDDEL ER OPNAADD I DENNE VASKEFASEN.
K2_V_DRIFT_OK 1310.00 BOOL
K2_V_RESET 1316.02 BOOL  ; 0-STILLER VASKEPGM.
K3_1_VMF_FERDIG 1326.00 BOOL
K3_COND_HJ1 923.05 BOOL
K3_DESINFEKSJON 1324.02 BOOL
K3_FASEFORLENG 1325.15 BOOL
K3_FASEF_OFFIMP 1326.06 BOOL  ; FERDIG-OFF-IMPULS.
K3_FEIL_LINJEPGM 1326.15 BOOL
K3_FORSINK_FEIL_FLOW T0234 BOOL
K3_FORSINK_SIRK T0180 BOOL
K3_FORSKYLL 1324.05 BOOL
K3_FORSK_LUT 1324.00 BOOL  ; FORSKYLL_LUT
K3_FORSK_LUT_DES 1324.01 BOOL  ; FORSKYLLING- LUT-DESINFEKSJON
K3_GRAFIKKTR_HJ1 921.08 BOOL
K3_GRM_FERDIG 1325.08 BOOL  ; GRENSEMELKFASEN AVSLUTTET.
K3_GRM_RESET 1326.04 BOOL
K3_GR_MELK_I_SYSTEM 1328.00 BOOL
K3_HJ1_TIL_TANK 1328.07 BOOL  ; ETTERRENNING_VED_TANKVASK
K3_HJ2_TIL_TANK_K3 1328.09 BOOL  ; ETTERRENNING_VED_TANKVASK
K3_HJ3_TIL_TANK_K3 1328.08 BOOL
K3_KONS_TID_FL 1327.00 BOOL
K3_LUT 1324.04 BOOL  ; LUT
K3_LUTVASK 1326.01 BOOL
K3_LUT_DES 1324.03 BOOL  ; LUT OG DESINFEKSJON
K3_LU_ER_STOERRE_PRS 1326.13 BOOL
K3_NOEDSTOPP 1325.05 BOOL  ; VASKEPROGR. STOPPER OG PUMPENE I VASKEN STOPPER.
K3_SIRKULASJON 1329.00 BOOL
K3_SPERR 1325.07 BOOL
K3_STERT_OK 1325.10 BOOL
K3_SY_ER_STOERRE_PRS 1326.14 BOOL
K3_TEMP_HJ1 923.06 BOOL
K3_TID_LL_TANK_S T0514 BOOL
K3_TID_LL_TANK_T 0514 NUMBER
K3_TR01_TID_S C0301 BOOL  ; KURS 3 TRINN 01 TID
K3_TR02_TID_S C0302 BOOL  ; KURS 3 TRINN 02 TID
K3_TR03_TID_PV C303 CHANNEL
K3_TR03_TID_S C0303 BOOL  ; KURS 3 TRINN 03 TID
K3_TR04_TID_S C0304 BOOL  ; KURS 3  TRINN 04 TID
K3_TR05_TID_S C0305 BOOL  ; KURS 3 TRINN 05 TID
K3_TR06_TID_S C0306 BOOL  ; KURS 3 TRINN 06 TID
K3_TR07_TID_PV C307 CHANNEL
K3_TR07_TID_S C0307 BOOL  ; KURS 3 TRINN 07 TID
K3_TR08_TID_S C0308 BOOL  ; KURS 3 TRINN 08 TID
K3_TR09_TID_S C0309 BOOL  ; KURS 3 TRINN 09 TID
K3_TR10_TID_S C0310 BOOL  ; KURS 3 TRINN 10 TID
K3_TR11_TID_S C0311 BOOL  ; KURS 3  TRINN 11 TID
K3_TR12_TID_S C0312 BOOL  ; KURS 3 TRINN 12 TID
K3_TR13_TID_S C0313 BOOL  ; KURS 3 TRINN 13 TID
K3_TR14_TID_S C0314 BOOL  ; KURS 3 TRINN 14 TID
K3_TR15_TID_S C0315 BOOL  ; KURS 3 TRINN 15 TID
K3_TR16_TID_S C0316 BOOL  ; KURS 3 TRINN 16 TID
K3_TR17_TID_S C0317 BOOL  ; KURS 3 TRINN 17 TID
K3_TR18_TID_S C0318 BOOL  ; KURS 3 TRINN 18 TID
K3_TR19_TID_S C0319 BOOL  ; KURS 3 TRINN 19 TID
K3_TR20_TID_S C0320 BOOL  ; KURS 3 TRINN 20 TID
K3_TR21_TID_PV C321 CHANNEL
K3_TR21_TID_S C0321 BOOL  ; KURS 3 TRINN 21 TID
K3_TR22_TID_S C0322 BOOL
K3_TR23_TID_S C0323 BOOL
K3_TR24_TID_S C0324 BOOL
K3_TR25_TID_S C0325 BOOL
K3_TR26_TID_S C0326 BOOL  ; KURS 3 TRINN 26 TID
K3_TR27_TID_S C0327 BOOL
K3_TR28_TID_S C0328 BOOL
K3_TR29_TID_S C0329 BOOL
K3_TR30_TID_S C0330 BOOL
K3_TRINNSKIFTE 1327.06 BOOL
K3_TURSTOPP 1325.13 BOOL  ; STANSER TURPUMPENE.
K3_TURTEMP_LAV 1329.01 BOOL
K3_TUR_HJ1 921.03 BOOL
K3_TUR_HJ2 921.04 BOOL
K3_TUR_HJ3 921.05 BOOL
K3_TUR_HJ4 921.06 BOOL
K3_VASK_INNE 1327.05 BOOL
K3_VENT_FOER_LUT 1329.02 BOOL
K3_VENT_TEMPERATUR 1329.03 BOOL
K3_VMFAS_RESET 1326.07 BOOL
K3_VM_KONOK 1325.09 BOOL  ; KONSENTRASJON-VASKEMIDDEL ER OPNAADD I DENNE VASKEFASEN.
K3_V_DRIFT_OK 1320.00 BOOL
K3_V_RESET 1326.02 BOOL  ; 0-STILLER VASKEPGM.
K4_SIST_LUT 1338.07 BOOL  ; SIST LUT TIL PASTEUR
K4_SIST_LUT_TID T0050 BOOL
K4_SIST_SYRE 1338.08 BOOL  ; SIST SYRE TIL PASTEUR
K4_SIST_SYRE_TID T0051 BOOL
KOMPULS1 993.08 BOOL
KOMPULS2 1994.09 BOOL
K_1_MINTEMP D8244 INT
K_2_MINTEMP D8246 INT
K_3_MINTEMP D8248 INT
L11_MELK_T03_VANN 712.06 BOOL
L11_MELK_T03_VANN_DRENERT 713.06 BOOL
L11_MELK_T04_VANN 712.07 BOOL
L11_MELK_T04_VANN_DRENERT 713.07 BOOL
L11_MELK_T05_VANN 712.08 BOOL
L11_MELK_T05_VANN_DRENERT 713.08 BOOL
L11_VANN_T03_MELK 712.01 BOOL
L11_VANN_T03_MELK_DRENERT 713.01 BOOL
L11_VANN_T03_VANN 712.00 BOOL
L11_VANN_T03_VANN_DRENERT 713.00 BOOL
L11_VANN_T04_MELK 712.03 BOOL
L11_VANN_T04_MELK_DRENERT 713.03 BOOL
L11_VANN_T04_VANN 712.02 BOOL
L11_VANN_T04_VANN_DRENERT 713.02 BOOL
L11_VANN_T05_MELK 712.05 BOOL
L11_VANN_T05_MELK_DRENERT 713.05 BOOL
L11_VANN_T05_VANN 712.04 BOOL
L11_VANN_T05_VANN_DRENERT 713.04 BOOL
L12_MELK_T03_VANN 714.06 BOOL
L12_MELK_T03_VANN_DRENERT 715.06 BOOL
L12_MELK_T04_VANN 714.07 BOOL
L12_MELK_T04_VANN_DRENERT 715.07 BOOL
L12_MELK_T05_VANN 714.08 BOOL
L12_MELK_T05_VANN_DRENERT 715.08 BOOL
L12_VANN_T03_MELK 714.01 BOOL
L12_VANN_T03_MELK_DRENERT 715.01 BOOL
L12_VANN_T03_VANN 714.00 BOOL
L12_VANN_T03_VANN_DRENERT 715.00 BOOL
L12_VANN_T04_MELK 714.03 BOOL
L12_VANN_T04_MELK_DRENERT 715.03 BOOL
L12_VANN_T04_VANN 714.02 BOOL
L12_VANN_T04_VANN_DRENERT 715.02 BOOL
L12_VANN_T05_MELK 714.05 BOOL
L12_VANN_T05_MELK_DRENERT 715.05 BOOL
L12_VANN_T05_VANN 714.04 BOOL
L12_VANN_T05_VANN_DRENERT 715.04 BOOL
L1_1_AUTODREN 701.00 BOOL  ; AUTODREN  L1.1
L1_1_BIL_AVSLUTTES 700.06 BOOL
L1_1_BIL_TOEMMES 700.05 BOOL
L1_1_DRENERER 700.08 BOOL
L1_1_DRENERT 700.12 BOOL  ; DRENERT KLAR TIL VASK
L1_1_DRENERT_RET H10.03 BOOL  ; HUSK STATUS
L1_1_DRENKONTR_TID_T 0690 NUMBER
L1_1_DRENSTART 700.07 BOOL
L1_1_DRENSTID_S T0043 BOOL
L1_1_DRENSTID_T 0043 NUMBER
L1_1_DREN_AVSL 700.09 BOOL
L1_1_DREN_M_REG_START 712.11 BOOL  ; REG.SIGNAL STARTMENGDE
L1_1_ER_MENGDE_DREN D2026 WORD  ; DRENERT MENGDE
L1_1_LINJETOEM_VASK 701.04 BOOL  ; TOEM LINJE ETTER VASK
L1_1_LINJETOEM_VASK_TID_C C0072 BOOL
L1_1_LINJETOEM_VASK_TID_S C72 CHANNEL
L1_1_MELK 700.11 BOOL  ; LINJE FYLT MED MELK
L1_1_MELK_RET H10.02 BOOL  ; HUSK STATUS
L1_1_MENGDE_RES 700.00 BOOL  ; RESET AV  TOTALMENGDE FOR LINJE
L1_1_SPERR 701.15 BOOL  ; SPERRER ALLE FUNKSJONER PAA LINJE. OGSAA VASK
L1_1_SPERRET_RET H10.05 BOOL
L1_1_SPERR_KODE_INN D2048 CHANNEL
L1_1_SPERR_KODE_UT D2049 CHANNEL
L1_1_ST_MENGDE_DREN D2024 WORD  ; REGISTRERT MENGDE VED START AV DREN.
L1_1_TMU_TID_S T0720 BOOL  ; INKOBLINGSTID TMU NAAR LINJE IKKE AKTIVERES
L1_1_TMU_TID_T 0720 NUMBER  ; MAX-TID TMU OM IKKE LINJE LEGGES
L1_1_UT_VANN_PRS D2028 WORD  ; PRS TOEMME LINJE FRA BIL TIL TANK FOR VANN
L1_1_V312_AAPEN 700.03 BOOL
L1_1_V312_LUKKER 700.04 BOOL
L1_1_VANN 700.10 BOOL
L1_1_VANN_DR_S T0680 BOOL
L1_1_VANN_DR_T 0680 NUMBER
L1_1_VANN_RET H10.01 BOOL  ; HUSK STATUS
L1_1_VANN_UT_DR_KT_TID_S T0690 BOOL
L1_1_VASKET 700.13 BOOL
L1_1_VASKET_RET H10.04 BOOL
L1_2_AUTODREN 703.00 BOOL  ; AUTODREN  L1.2
L1_2_BIL_AVSLUTTES 702.06 BOOL
L1_2_BIL_TOEMMES 702.05 BOOL
L1_2_C81_CONTAINER 1309.06 BOOL
L1_2_DRENERER 702.08 BOOL
L1_2_DRENERT 702.12 BOOL  ; DRENERT KLAR TIL VASK
L1_2_DRENERT_RET H11.03 BOOL  ; HUSK STATUS
L1_2_DRENKONTR_TID_T 0691 NUMBER
L1_2_DRENSTART 702.07 BOOL
L1_2_DRENSTID_S T0044 BOOL
L1_2_DRENSTID_T 0044 NUMBER
L1_2_DREN_AVSL 702.09 BOOL
L1_2_ER_MENGDE_DREN D2126 WORD  ; DRENERT MENGDE
L1_2_LINJETOEM_VASK 703.04 BOOL  ; TOEM LINJE ETTER VASK
L1_2_LINJETOEM_VASK_TID_C C0073 BOOL
L1_2_LINJETOEM_VASK_TID_S C73 CHANNEL
L1_2_MELK 702.11 BOOL  ; LINJE FYLT MED MELK
L1_2_MELK_RET H11.02 BOOL  ; HUSK STATUS
L1_2_MENGDE_RES 702.00 BOOL  ; RESET AV  TOTALMENGDE FOR LINJE
L1_2_SPERR 703.15 BOOL  ; SPERRER ALLE FUNKSJONER PAA LINJE. OGSAA VASK
L1_2_SPERRET_RET H11.05 BOOL
L1_2_SPERR_KODE_INN D2148 CHANNEL
L1_2_SPERR_KODE_UT D2149 CHANNEL
L1_2_ST_MENGDE_DREN D2124 WORD  ; REGISTRERT MENGDE VED START AV DREN.
L1_2_TMU 521.08 BOOL  ; TILBAKEMELDINGSUTK0BLING
L1_2_TMU_TID_S T0721 BOOL  ; INKOBLINGSTID TMU NAAR LINJE IKKE AKTIVERES
L1_2_TMU_TID_T 0721 NUMBER  ; MAX-TID TMU OM IKKE LINJE LEGGES
L1_2_UT_VANN_PRS D2128 WORD  ; PRS TOEMME LINJE FRA BIL TIL TANK FOR VANN
L1_2_V322_AAPEN 702.03 BOOL
L1_2_V322_LUKKER 702.04 BOOL
L1_2_VANN 702.10 BOOL
L1_2_VANN_DR_S T0681 BOOL
L1_2_VANN_DR_T 0681 NUMBER
L1_2_VANN_RET H11.01 BOOL
L1_2_VANN_UT_DR_KT_TID_S T0691 BOOL
L1_2_VASKET 702.13 BOOL
L1_2_VASKET_RET H11.04 BOOL  ; HUSK STATUS
L1_TOT_MENGDE D2402 WORD  ; SUM L1.1 OG L1.2
L21_MELK_T03_VANN 716.06 BOOL
L21_MELK_T03_VANN_DRENERT 717.06 BOOL
L21_MELK_T04_VANN 716.07 BOOL
L21_MELK_T04_VANN_DRENERT 717.07 BOOL
L21_MELK_T05_VANN 716.08 BOOL
L21_MELK_T05_VANN_DRENERT 717.08 BOOL
L21_VANN_T03_MELK 716.01 BOOL
L21_VANN_T03_MELK_DRENERT 717.01 BOOL
L21_VANN_T03_VANN 716.00 BOOL
L21_VANN_T03_VANN_DRENERT 717.00 BOOL
L21_VANN_T04_MELK 716.03 BOOL
L21_VANN_T04_MELK_DRENERT 717.03 BOOL
L21_VANN_T04_VANN 716.02 BOOL
L21_VANN_T04_VANN_DRENERT 717.02 BOOL
L21_VANN_T05_MELK 716.05 BOOL
L21_VANN_T05_MELK_DRENERT 717.05 BOOL
L21_VANN_T05_VANN 716.04 BOOL
L21_VANN_T05_VANN_DRENERT 717.04 BOOL
L22_MELK_T03_VANN 718.06 BOOL
L22_MELK_T03_VANN_DRENERT 719.06 BOOL
L22_MELK_T04_VANN 718.07 BOOL
L22_MELK_T04_VANN_DRENERT 719.07 BOOL
L22_MELK_T05_VANN 718.08 BOOL
L22_MELK_T05_VANN_DRENERT 719.08 BOOL
L22_VANN_T03_MELK 718.01 BOOL
L22_VANN_T03_MELK_DRENERT 719.01 BOOL
L22_VANN_T03_VANN 718.00 BOOL
L22_VANN_T03_VANN_DRENERT 719.00 BOOL
L22_VANN_T04_MELK 718.03 BOOL
L22_VANN_T04_MELK_DRENERT 719.03 BOOL
L22_VANN_T04_VANN 718.02 BOOL
L22_VANN_T04_VANN_DRENERT 719.02 BOOL
L22_VANN_T05_MELK 718.05 BOOL
L22_VANN_T05_MELK_DRENERT 719.05 BOOL
L22_VANN_T05_VANN 718.04 BOOL
L22_VANN_T05_VANN_DRENERT 719.04 BOOL
L2_1_AUTODREN 705.00 BOOL  ; AUTODREN  L2.1
L2_1_BIL_AVSLUTTES 704.06 BOOL
L2_1_BIL_TOEMMES 704.05 BOOL
L2_1_DRENERER 704.08 BOOL
L2_1_DRENERT 704.12 BOOL  ; DRENERT KLAR TIL VASK
L2_1_DRENERT_RET H12.03 BOOL  ; HUSK STATUS
L2_1_DRENKONTR_TID_T 0692 NUMBER
L2_1_DRENSTART 704.07 BOOL
L2_1_DRENSTID_S T0045 BOOL
L2_1_DRENSTID_T 0045 NUMBER
L2_1_DREN_AVSL 704.09 BOOL
L2_1_ER_MENGDE_DREN D2226 WORD  ; DRENERT MENGDE
L2_1_LINJETOEM_VASK 705.04 BOOL  ; TOEM LINJE ETTER VASK
L2_1_LINJETOEM_VASK_TID_C C0074 BOOL
L2_1_LINJETOEM_VASK_TID_S C74 CHANNEL
L2_1_MELK 704.11 BOOL  ; LINJE FYLT MED MELK
L2_1_MELK_RET H12.02 BOOL  ; HUSK STATUS
L2_1_MENGDE_RES 704.00 BOOL  ; RESET AV  TOTALMENGDE FOR LINJE
L2_1_SPERR 705.15 BOOL  ; SPERRER ALLE FUNKSJONER PAA LINJE. OGSAA VASK
L2_1_SPERRET_RET H12.05 BOOL
L2_1_SPERR_KODE_INN D2248 CHANNEL
L2_1_SPERR_KODE_UT D2249 CHANNEL
L2_1_ST_MENGDE_DREN D2224 WORD  ; REGISTRERT MENGDE VED START AV DREN.
L2_1_TMU 522.08 BOOL  ; TILBAKEMELDINGSUTK0BLING
L2_1_TMU_TID_S T0722 BOOL  ; INKOBLINGSTID TMU NAAR LINJE IKKE AKTIVERES
L2_1_TMU_TID_T 0722 NUMBER  ; MAX-TID TMU OM IKKE LINJE LEGGES
L2_1_UT_VANN_PRS D2228 WORD  ; PRS TOEMME LINJE FRA BIL TIL TANK FOR VANN
L2_1_V332_AAPEN 704.03 BOOL
L2_1_VANN 704.10 BOOL
L2_1_VANN_DR_S T0684 BOOL
L2_1_VANN_DR_T 0684 NUMBER
L2_1_VANN_RET H12.01 BOOL  ; HUSK STATUS
L2_1_VANN_UT_DR_KT_TID_S T0692 BOOL
L2_1_VASKET 704.13 BOOL
L2_1_VASKET_RET H12.04 BOOL  ; HUSK STATUS
L2_2_AUTODREN 707.00 BOOL  ; AUTODREN  L2.2
L2_2_BIL_AVSLUTTES 706.06 BOOL
L2_2_BIL_TOEMMES 706.05 BOOL
L2_2_DRENERER 706.08 BOOL
L2_2_DRENERT 706.12 BOOL  ; DRENERT KLAR TIL VASK
L2_2_DRENERT_RET H13.03 BOOL  ; HUSK STATUS
L2_2_DRENKONTR_TID_T 0693 NUMBER
L2_2_DRENSTART 706.07 BOOL
L2_2_DRENSTID_S T0046 BOOL
L2_2_DRENSTID_T 0046 NUMBER
L2_2_DREN_AVSL 706.09 BOOL
L2_2_ER_MENGDE_DREN D2326 WORD  ; DRENERT MENGDE
L2_2_LINJETOEM_VASK 707.04 BOOL  ; TOEM LINJE ETTER VASK
L2_2_LINJETOEM_VASK_TID_C C0075 BOOL
L2_2_LINJETOEM_VASK_TID_S C75 CHANNEL
L2_2_MELK 706.11 BOOL  ; LINJE FYLT MED MELK
L2_2_MELK_RET H13.02 BOOL  ; HUSK STATUS
L2_2_MENGDE_RES 706.00 BOOL  ; RESET AV  TOTALMENGDE FOR LINJE
L2_2_SPERR 707.15 BOOL  ; SPERRER ALLE FUNKSJONER PAA LINJE. OGSAA VASK
L2_2_SPERRET_RET H13.05 BOOL
L2_2_SPERR_KODE_INN D2348 CHANNEL
L2_2_SPERR_KODE_UT D2349 CHANNEL
L2_2_ST_MENGDE_DREN D2324 WORD  ; REGISTRERT MENGDE VED START AV DREN.
L2_2_TMU 523.08 BOOL  ; TILBAKEMELDINGSUTKOBLING
L2_2_TMU_TID_S T0723 BOOL  ; INKOBLINGSTID TMU NAAR LINJE IKKE AKTIVERES
L2_2_TMU_TID_T 0723 NUMBER  ; MAX-TID TMU OM IKKE LINJE LEGGES
L2_2_UT_VANN_PRS D2328 WORD  ; PRS TOEMME LINJE FRA BIL TIL TANK FOR VANN
L2_2_V342_AAPEN 706.03 BOOL
L2_2_VANN 706.10 BOOL
L2_2_VANN_DR_S T0685 BOOL
L2_2_VANN_DR_T 0685 NUMBER
L2_2_VANN_RET H13.01 BOOL  ; HUSK STATUS
L2_2_VANN_UT_DR_KT_TID_S T0693 BOOL
L2_2_VASKET 706.13 BOOL
L2_2_VASKET_RET H13.04 BOOL  ; HUSK STATUS
L2_TOT_MENGDE D2404 WORD  ; SUM L2.1 OG L2.2
L3_DRENERT 708.10 BOOL
L3_DRENERT_RET H20.02 BOOL  ; HUSK STATUS
L3_DREN_PAST21_IND 1226.00 BOOL
L3_DREN_PAST22_IND 1227.00 BOOL
L3_PRODUKT_PAST21_IND 1226.02 BOOL  ; INDIVIDADR
L3_PRODUKT_PAST22_IND 1227.02 BOOL  ; INDIVIDADR
L3_SPERR 709.15 BOOL  ; SPERRER ALLE FUNKSJONER PAA LINJE. OGSAA VASK
L3_SPERRET_HR H20.03 BOOL
L3_VASKET 708.13 BOOL
L3_VASKET_RET H20.01 BOOL  ; HUSK STATUS
L4_DRENERT 710.10 BOOL
L4_DRENERT_RET H21.02 BOOL  ; HUSK STATUS
L4_DREN_PAST21_IND 1226.01 BOOL  ; INDIVIDADR
L4_DREN_PAST22_IND 1227.01 BOOL  ; INDIVIDADR
L4_PRODUKT_PAST21_IND 1226.03 BOOL  ; INDIVIDADR
L4_PRODUKT_PAST22_IND 1227.03 BOOL  ; INDIVIDADR
L4_SPERR 711.15 BOOL  ; SPERRER ALLE FUNKSJONER PAA LINJE. OGSAA VASK
L4_SPERRET_HR H21.03 BOOL
L4_VASKET 710.13 BOOL
L4_VASKET_RET H21.01 BOOL  ; HUSK STATUS
LAMPE_L1_2_C81_CONTAINER 2100.04 BOOL
LAMPE_LAB_HJ 960.07 BOOL
LINJEKOMMANDO D3000 CHANNEL
LL_BLK21 4500.15 BOOL
LL_BLK22 4510.15 BOOL
LL_BLK23 4520.15 BOOL
LL_BLK23_UREN 4522.00 BOOL  ; D_VITAMIN
LL_T03 600.01 BOOL
LL_T03_FORSINKELSE T0611 BOOL  ; TID SOM FORSINKER  BUNNVARSEL PAA T03
LL_T03_PLS1 4600.01 BOOL
LL_T04 602.01 BOOL
LL_T04_PLS1 4600.03 BOOL
LL_T04_SPERRE 602.02 BOOL  ; RESETTER  LL OG SPERRER LL TID  VED FYLLING AV TANK
LL_T05 604.01 BOOL
LL_T05_PLS1 4600.05 BOOL
LL_T05_SPERRE 604.02 BOOL  ; RESETTER  LL OG SPERRER LL TID  VED FYLLING AV TANK
LL_T24_01 750.01 BOOL
LL_T24_01_FORSINKELSE_S T0669 BOOL  ; TID SOM FORSINKER  BUNNVARSEL PAA T24.01
LL_T24_01_FORSINKELSE_T 0669 NUMBER  ; BUNJNVARSEL PAA T24.01
LL_T2701 688.01 BOOL
LL_T2702 689.01 BOOL
LL_T2703 690.01 BOOL
LL_T40 648.01 BOOL
LL_T40_FORSINKELSE_S T0613 BOOL  ; TID SOM FORSINKER  BUNNVARSEL PAA T40
LL_T40_FORSINKELSE_T 0613 NUMBER  ; TID SOM FORSINKER  BUNNVARSEL PAA T40
LL_T41 649.01 BOOL
LL_T41_FORSINKELSE_S T0615 BOOL  ; TID SOM FORSINKER  BUNNVARSEL PAA T41
LL_T41_FORSINKELSE_T 0615 NUMBER  ; TID SOM FORSINKER  BUNNVARSEL PAA T41
LL_T81 1401.11 BOOL
LL_T82 1402.11 BOOL  ; LL- T 82 Luttank.
LL_T83 1403.11 BOOL  ; LL- T 83 Syretank.
LL_T84 1404.11 BOOL  ; LL- T 84 Hetvanntank.
LOW_LEVEL_BLK21 LOW_LEVEL
LOW_LEVEL_BLK22 LOW_LEVEL
LOW_LEVEL_BLK23 HIGH_LEVEL
LUKK_V8036 1000.06 BOOL
LUKK_V8037 1000.07 BOOL
LUKK_V8043 1000.08 BOOL
M2111_AUTO 1055.03 BOOL  ; MOTOR HOMOGENISATOR 21
M2111_INN 2702.03 BOOL  ; MOTOR HOMOGENISATOR 21
M2111_MAN 1005.03 BOOL  ; MOTOR HOMOGENISATOR 21
M2111_UT 2402.03 BOOL  ; MOTOR HOMOGENISATOR 21
M2211_AUTO 1056.11 BOOL
M2211_INN 2701.15 BOOL  ; MOTOR HOMOGENISATOR 22
M2211_MAN 1006.11 BOOL
M2211_UT 2401.15 BOOL  ; ¨
M2301_1_INN 2704.05 BOOL  ; KJOELEVIFTE P2301
MANUELL_KOMMAND D3002 CHANNEL  ; KOMMANDOORD FOR IKKE LINJEKOMMANDOER
MAN_DAMP_T82 1402.03 BOOL
MAN_DAMP_T83 1403.03 BOOL
MAN_DESINF_T84 1404.04 BOOL
MAN_DOS_T82 1402.02 BOOL  ; Manuell Doser vaskemiddel. T 82 Luttank.
MAN_DOS_T83 1403.02 BOOL  ; Manuell Doser vaskemiddel. T 83 Syretank.
MAN_DOS_T84 1404.02 BOOL
MAN_FYLL_V_T81 1401.01 BOOL  ; Manuell fyll vann. T 81 Forskylletank.
MAN_FYLL_V_T82 1402.01 BOOL  ; Manuell fyll vann. T 82 Luttank.
MAN_FYLL_V_T83 1403.01 BOOL  ; Manuell fyll vann. T 83 Syretank.
MAN_FYLL_V_T84 1404.01 BOOL  ; Manuell fyll vann. T 84 Hetvanntank.
MAN_LUT_T82 1402.04 BOOL
MAN_SYRE_T83 1403.04 BOOL
MAN_V4550_COM_BIT 1150.04 BOOL  ; VANNVENTIL V4550 UTGJEVNINGSBEHOLDER 27.45  MANUELT
MAN_V4550_TID T0001 BOOL  ; VANNVENTIL V4550 UTGJEVNINGSBEHOLDER 27.45  MANUELT
MIXTANKER_SLUK 723.08 BOOL  ; T20.11-19 TIL SLUK
MIX_D_FOR 698.03 BOOL  ; T20.11-19  TIL T27.40-41. P1940 STARTER
MIX_D_SLUK 698.04 BOOL
MIX_M3_COMAND_ORD 2914 WORD  ; FRA T20.11-19                                                      1=SLUK                                                                     2=DYREFOR
MOTTAK_TOT_MENGDE D2400 WORD
MOT_AUTODR_DAG_PRS D1981 REAL
MOT_AUTODR_MAANED_PRS D1980 REAL
MOT_AUTODR_MIN_PRS D1983 REAL
MOT_AUTODR_START 698.01 BOOL  ; AUTODREN FOR ALLE LINJER IMOTTAGELSEN STARTES FRA GRAFIKK
MOT_AUTODR_TIME_PRS D1982 REAL
MOT_AUTODR_VALGT 698.00 BOOL  ; AUTODREN FOR ALLE LINJER IMOTTAGELSEN VALGT
MOXERTANK_D_FOR 723.09 BOOL  ; TIL TANK TIL T27.40-41
N4_DRIFT 2000.00 BOOL  ; NODE4 STARTET OG INNE
N4_PGM552_0_STATUS 2810.09 BOOL
N4_PGM552_1_STATUS 2810.10 BOOL
N5_0644_INN 2923.04 BOOL
N5_90K1_KL_TRINN 2906 CHANNEL
N5_90K2_KL_TRINN 2907 CHANNEL
N5_90K3_KL_TRINN 2908 CHANNEL
N5_B4201_SLANGKONTR 2980.06 BOOL  ; SLANGEKONTROLL VED TRAKT T27.42
N5_DRN_T2013_TIL_FORTANK 2932.01 BOOL
N5_DRN_T2013_TIL_SLUK 2932.02 BOOL
N5_DRN_T2013_TIL_UHT 2932.03 BOOL
N5_DRN_T2014_TIL_FORTANK 2932.06 BOOL
N5_DRN_T2014_TIL_SLUK 2932.07 BOOL
N5_DRN_T2014_TIL_UHT 2932.08 BOOL
N5_DRN_T2015_TIL_FORTANK 2932.11 BOOL
N5_DRN_T2015_TIL_SLUK 2932.12 BOOL
N5_DRN_T2015_TIL_UHT 2932.13 BOOL
N5_DRN_T2016_TIL_FORTANK 2933.01 BOOL
N5_DRN_T2016_TIL_SLUK 2933.02 BOOL
N5_DRN_T2016_TIL_UHT 2933.03 BOOL
N5_DRN_T2017_TIL_FORTANK 2933.06 BOOL
N5_DRN_T2017_TIL_SLUK 2933.07 BOOL
N5_DRN_T2017_TIL_UHT 2933.08 BOOL
N5_DRN_T2018_DRIFT 2933.10 BOOL
N5_DRN_T2018_TIL_FORTANK 2933.11 BOOL
N5_DRN_T2018_TIL_SLUK 2933.12 BOOL
N5_DRN_T2018_TIL_UHT 2933.13 BOOL
N5_DRN_T2019_TIL_FORTANK 2934.01 BOOL
N5_DRN_T2019_TIL_SLUK 2934.02 BOOL
N5_DRN_T2019_TIL_UHT 2934.03 BOOL
N5_P1101_PAADRAG 2939 CHANNEL  ; 0-1000 TIL NODE 2.17
N5_P1101_UT 2938.14 BOOL  ; TIL NODE 2.17
N5_P1102_UT 2938.15 BOOL  ; TIL NODE 2.17
N5_P1940_U 2903.05 BOOL  ; UHT AVD
N5_P2021_U 2903.06 BOOL  ; UHT AVD
N5_P2027_INN 2819.06 BOOL
N5_P2027_U 2903.07 BOOL  ; UHT AVD
N5_P2039_UT 2904.03 BOOL
N5_P2060_STARTSIGNAL 2900.11 BOOL
N5_PANEL19_P2060_START 2903.00 BOOL  ; RELE 19K101 I PANEL 19 ( 7-8M3 PANEL)
N5_PG541_DRIFT 2901.01 BOOL
N5_PG542_DRIFT 2901.08 BOOL
N5_PGM501_0_STATUS 2924.02 BOOL
N5_PGM501_1_STATUS 2924.03 BOOL
N5_PGM501_2_STATUS 2924.04 BOOL
N5_PGM501_DRIFT 2924.01 BOOL
N5_PGM501_IKKE_FEIL 2924.05 BOOL
N5_PGM501_STOPP 2924.00 BOOL
N5_PGM505_0_STATUS 2926.02 BOOL
N5_PGM505_1_STATUS 2926.03 BOOL
N5_PGM505_2_STATUS 2926.04 BOOL
N5_PGM505_DRIFT 2926.01 BOOL
N5_PGM505_IKKE_FEIL 2926.05 BOOL
N5_PGM505_STOPP 2926.00 BOOL
N5_PGM510_0_STAT 2902.06 BOOL
N5_PGM510_1_STAT 2902.07 BOOL
N5_PGM510_2_STAT 2902.08 BOOL
N5_PGM510_IKKE_FEIL 2902.09 BOOL  ; 1 = ER IKKE FEIL
N5_PGM510_IND_C26 2900.03 BOOL  ; T20.02
N5_PGM510_IND_C27 2900.04 BOOL  ; T20.33 (03)
N5_PGM510_IND_C28 2900.05 BOOL  ; T20.34 (04)
N5_PGM510_IND_C29 2900.06 BOOL  ; T20.35 (05)
N5_PGM510_IND_C80 2900.02 BOOL  ; RV T20.28-T20.29
N5_PGM510_IND_C87 2900.07 BOOL
N5_PGM510_IND_C88 2900.08 BOOL  ; T20.30 SCANIMA
N5_PGM510_IND_C89 2900.09 BOOL
N5_PGM510_IND_C90 2900.00 BOOL  ; T20.28
N5_PGM510_IND_C91 2900.01 BOOL  ; T20.29
N5_PGM510_IND_C92 2900.10 BOOL  ; RV STERIL
N5_PGM510_TMU_N4 2905.14 BOOL
N5_PGM511_0_STAT 2931.06 BOOL
N5_PGM511_1_STAT 2931.07 BOOL
N5_PGM511_2_STAT 2931.08 BOOL
N5_PGM511_IKKE_FEIL 2931.09 BOOL  ; 1 = ER IKKE FEIL
N5_PGM511_IND_C39 2901.00 BOOL  ; T20.11
N5_PGM511_IND_C40 2901.01 BOOL  ; T20.12
N5_PGM511_IND_C41 2901.02 BOOL  ; T20.14
N5_PGM511_IND_C43 2901.04 BOOL  ; T20.16
N5_PGM511_IND_C44 2901.05 BOOL  ; T20.15
N5_PGM511_IND_C45 2901.06 BOOL  ; RV
N5_PGM511_IND_C47 2901.07 BOOL
N5_PGM511_IND_C49 2901.09 BOOL  ; RV
N5_PGM511_IND_C57 2901.10 BOOL  ; T20.18
N5_PGM511_IND_C58 2901.11 BOOL  ; T20.17
N5_PGM511_IND_C93 2901.12 BOOL  ; T20.36
N5_PGM511_IND_C94 2901.13 BOOL  ; T20.37
N5_PGM512_0_STAT 2934.06 BOOL
N5_PGM512_1_STAT 2934.07 BOOL
N5_PGM512_2_STAT 2934.08 BOOL
N5_PGM512_IKKE_FEIL 2934.09 BOOL  ; 1 = ER IKKE FEIL
N5_PGM512_IND_C55 2931.11 BOOL  ; TV-STERIL
N5_PGM512_IND_C56 2931.12 BOOL  ; RV-STERIL
N5_PGM515_0_STATUS 2954.10 BOOL
N5_PGM515_1_STATUS 2954.11 BOOL
N5_PGM515_2_STATUS 2954.12 BOOL
N5_PGM515_IKKE_FEIL 2954.13 BOOL
N5_PGM515_IND_C16 2954.00 BOOL
N5_PGM515_IND_C17 2954.01 BOOL
N5_PGM515_IND_C18 2954.02 BOOL
N5_PGM515_IND_C19 2954.03 BOOL
N5_PGM515_IND_C20 2954.04 BOOL
N5_PGM515_IND_C21 2954.07 BOOL
N5_PGM515_IND_C22 2954.05 BOOL
N5_PGM515_IND_C46 2954.08 BOOL
N5_PGM515_IND_C76 2954.06 BOOL
N5_PGM515_TMU 2954.14 BOOL
N5_PGM530_0_STATUS 2930.00 BOOL  ; PAST21 TIL UHT
N5_PGM530_1_STATUS 2930.01 BOOL  ; PAST21 TIL UHT
N5_PGM530_2_STAT 2930.02 BOOL  ; PAST21 TIL UHT
N5_PGM530_DIREKTE_IND 2920.04 BOOL
N5_PGM530_IKKE_FEIL 2930.03 BOOL  ; PAST21 TIL UHT
N5_PGM530_KOE_DR 2902.12 BOOL
N5_PGM530_T2009_IND 2920.00 BOOL
N5_PGM530_T2033_IND 2920.01 BOOL
N5_PGM530_T2034_IND 2920.02 BOOL
N5_PGM530_T2035_IND 2920.03 BOOL
N5_PGM531_0_STATUS 2930.06 BOOL  ; PAST22 TIL UHT
N5_PGM531_1_STATUS 2930.07 BOOL  ; PAST22 TIL UHT
N5_PGM531_2_STAT 2930.08 BOOL  ; PAST22 TIL UHT
N5_PGM531_DIREKTE_IND 2920.09 BOOL
N5_PGM531_IKKE_FEIL 2930.09 BOOL  ; PAST22 TIL UHT
N5_PGM531_KOE_DR 2902.11 BOOL
N5_PGM531_T2033_IND 2920.06 BOOL
N5_PGM531_T2034_IND 2920.07 BOOL
N5_PGM531_T2035_IND 2920.08 BOOL
N5_PGM532_0_STATUS 2930.11 BOOL  ; PAST23 TIL UHT
N5_PGM532_1_STATUS 2930.12 BOOL  ; PAST23 TIL UHT
N5_PGM532_2_STAT 2930.13 BOOL  ; PAST23 TIL UHT
N5_PGM532_DIREKTE_IND 2920.14 BOOL
N5_PGM532_IKKE_FEIL 2930.14 BOOL  ; PAST22 TIL UHT
N5_PGM532_T2033_IND 2920.11 BOOL
N5_PGM532_T2034_IND 2920.12 BOOL
N5_PGM532_T2035_IND 2920.13 BOOL
N5_PGM541_1_STAT 2901.03 BOOL
N5_PGM546_0_STATUS 2931.00 BOOL
N5_PGM546_1_STATUS 2931.01 BOOL
N5_PGM546_2_STAT 2931.02 BOOL
N5_PGM546_IKKE_FEIL 2931.03 BOOL
N5_PGM546_T2009_DREN_IND 2921.01 BOOL  ; DREN FRA V2347
N5_PGM546_T2009_IND 2921.00 BOOL
N5_PGM552_0_STATUS 2926.08 BOOL
N5_PGM552_1_STATUS 2926.09 BOOL
N5_PGM552_2_STATUS 2926.10 BOOL
N5_PGM552_IKKE_FEIL 2917.14 BOOL  ; PAST21 TIL T.GR08 OG T20.28-29
N5_PGM552_IND_P21_T0801 2924.08 BOOL
N5_PGM552_IND_P21_T0802 2924.09 BOOL
N5_PGM552_IND_P21_T0803 2924.10 BOOL
N5_PGM552_IND_P21_T0804 2924.11 BOOL
N5_PGM552_IND_P21_T0805 2924.12 BOOL
N5_PGM552_IND_P21_T2028 2924.13 BOOL
N5_PGM552_IND_P21_T2029 2924.14 BOOL
N5_PGM552_TMU 2926.12 BOOL
N5_PGM552_iKKE_FEIL 2926.11 BOOL
N5_PGM553_0_STATUS 2948.05 BOOL  ; 0_STATUS!
N5_PGM553_1_STATUS 2948.06 BOOL  ; 1_STATUS!
N5_PGM553_2_STATUS 2948.07 BOOL  ; 2_STATUS!
N5_PGM553_IKKE_FEIL 2948.08 BOOL
N5_PGM553_IND_P21_T0901 2948.00 BOOL
N5_PGM553_IND_P21_T0902 2948.01 BOOL
N5_PGM553_IND_P21_T0903 2948.02 BOOL
N5_PGM553_IND_P21_T0904 2948.03 BOOL
N5_PGM553_IND_P21_T0905 2948.04 BOOL
N5_PGM553_TMU 2948.09 BOOL
N5_PGM554_0_STATUS 2947.08 BOOL
N5_PGM554_1_STATUS 2947.09 BOOL
N5_PGM554_2_STATUS 2947.10 BOOL
N5_PGM554_IKKE_FEIL 2947.11 BOOL
N5_PGM554_IND_P22_T0801 2947.00 BOOL
N5_PGM554_IND_P22_T0802 2947.01 BOOL
N5_PGM554_IND_P22_T0803 2947.02 BOOL
N5_PGM554_IND_P22_T0804 2947.03 BOOL
N5_PGM554_IND_P22_T0805 2947.04 BOOL
N5_PGM554_IND_P22_T2028 2947.05 BOOL
N5_PGM554_IND_P22_T2029 2947.06 BOOL
N5_PGM554_TMU 2947.12 BOOL
N5_PGM555_0_STATUS 2949.06 BOOL  ; 0_STATUS!
N5_PGM555_1_STATUS 2949.07 BOOL  ; 1_STATUS!
N5_PGM555_2_STATUS 2949.08 BOOL  ; 2_STATUS!
N5_PGM555_IKKE_FEIL 2949.09 BOOL  ; 1=IKKE FEIL
N5_PGM555_IND_P22_T0901 2949.00 BOOL
N5_PGM555_IND_P22_T0902 2949.01 BOOL
N5_PGM555_IND_P22_T0903 2949.02 BOOL
N5_PGM555_IND_P22_T0904 2949.03 BOOL
N5_PGM555_IND_P22_T0905 2949.04 BOOL
N5_PGM555_IND_P22_TGR11 2949.05 BOOL
N5_PGM555_TMU 2949.10 BOOL
N5_PGM556_0_STATUS 2953.04 BOOL  ; 0_STATUS!
N5_PGM556_1_STATUS 2953.05 BOOL  ; 1_STATUS!
N5_PGM556_2_STATUS 2953.06 BOOL  ; 2_STATUS!
N5_PGM556_IKKE_FEIL 2953.07 BOOL
N5_PGM556_IND_P23_DREN 2953.03 BOOL
N5_PGM556_IND_P23_T1002 2953.00 BOOL
N5_PGM556_IND_P23_T1003 2953.01 BOOL
N5_PGM556_IND_P23_T1004 2953.02 BOOL
N5_PGM556_TMU 2953.08 BOOL
N5_PGM558_DIREKTE_IND 2935.03 BOOL
N5_PGM558_T2033_IND 2935.00 BOOL
N5_PGM558_T2034_IND 2935.01 BOOL
N5_PGM558_T2035_IND 2935.02 BOOL
N5_PGM559_0_STATUS 2925.01 BOOL
N5_PGM559_1_STATUS 2925.02 BOOL
N5_PGM559_2_STATUS 2925.03 BOOL
N5_PGM559_DREN_IND 2925.00 BOOL
N5_PGM559_IKKE_FEIL 2925.04 BOOL
N5_PGM559_TMU 2925.05 BOOL
N5_PGM560_0_STATUS 2925.09 BOOL
N5_PGM560_1_STATUS 2925.10 BOOL
N5_PGM560_2_STATUS 2925.11 BOOL
N5_PGM560_IKKE_FEIL 2925.12 BOOL
N5_PGM560_P22_TIL_RETURT_IND 2925.08 BOOL
N5_PGM560_TMU 2925.13 BOOL
N5_PGM561_0_STATUS 2922.01 BOOL
N5_PGM561_1_STATUS 2922.02 BOOL
N5_PGM561_2_STATUS 2922.03 BOOL
N5_PGM561_IKKE_FEIL 2922.04 BOOL  ; ¨
N5_PGM561_P21_TIL_T2009_IND 2922.00 BOOL
N5_PGM561_TMU 2922.05 BOOL
N5_PGM562_0_STATUS 2922.09 BOOL  ; ¨
N5_PGM562_1_STATUS 2922.10 BOOL
N5_PGM562_2_STAT 2922.11 BOOL
N5_PGM562_IKKE_FEIL 2922.12 BOOL  ; 1= IKKE FEIL
N5_PGM562_IND_T2009 2922.08 BOOL
N5_Q2022_OPN_FORV 2901.14 BOOL
N5_R20_36_02_SERVICEBR 2902.03 BOOL  ; 1=OK
N5_R20_37_02_SERVICEBR 2902.04 BOOL  ; 1=OK
N5_RV2013_01_HOEY_UT 2921.04 BOOL  ; HOEY HASTIGHET
N5_RV2013_01_LAV_UT 2921.03 BOOL  ; LAV HASTIGHET
N5_RV2013_02_UT 2921.05 BOOL
N5_RV2014_01_HOEY_UT 2921.07 BOOL  ; HOEY HASTIGHET
N5_RV2014_01_LAV_UT 2921.06 BOOL
N5_RV2014_02_UT 2921.08 BOOL
N5_RV2036_NIVSTOP 2921.14 BOOL
N5_RV2037_NIVSTOP 2921.13 BOOL
N5_RV20_11_01_U 2917.05 BOOL  ; T20.11 UHT AVD
N5_RV20_12_01_U 2917.06 BOOL  ; T20.12 UHT AVD
N5_RV20_17_01_U 2919.12 BOOL  ; T20.17 UHT AVD
N5_RV20_33_01_U 2917.00 BOOL  ; T20.33 UHT AVD
N5_RV20_34_01_U 2917.01 BOOL  ; T20.34 UHT AVD
N5_RV20_35_01_U 2917.02 BOOL  ; T20.35 UHT AVD
N5_SLC500NY_C45_INNKOBLET 2903.01 BOOL  ; TIL SLC
N5_SLC500NY_LINJE_P2029_OK 2903.02 BOOL  ; TIL SLC
N5_SLC500_PRODUKT_INNE 2918.14 BOOL  ; PRODUKT FRA T20.11 TIL 20.37 ER INNKOBLET
N5_T2009_PT 2960 INT
N5_T2009_TT 2959 INT
N5_T2011_MANUELL_AAPNING 2936.03 BOOL
N5_T2011_PT 2962 INT
N5_T2011_TT 2961 INT
N5_T2012_MANUELL_AAPNING 2936.04 BOOL
N5_T2012_PT 2964 INT
N5_T2012_TT 2963 INT
N5_T2013_MANUELL_AAPNING 2936.05 BOOL
N5_T2013_PT 2966 INT
N5_T2013_TT 2965 INT
N5_T2014_MANUELL_AAPNING 2936.06 BOOL
N5_T2014_PT 2968 INT
N5_T2014_TT 2967 INT
N5_T2015_MANUELL_AAPNING 2936.07 BOOL
N5_T2015_PT 2970 INT
N5_T2015_TT 2969 INT
N5_T2016_MANUELL_AAPNING 2936.08 BOOL
N5_T2016_PT 2972 INT
N5_T2016_TT 2971 INT
N5_T2017_MANUELL_AAPNING 2936.09 BOOL
N5_T2017_PT 2974 INT
N5_T2017_TT 2973 INT
N5_T2018_MANUELL_AAPNING 2936.10 BOOL
N5_T2018_PT 2976 INT
N5_T2018_TT 2975 INT
N5_T2019_MANUELL_AAPNING 2936.11 BOOL
N5_T2019_PT 2978 INT
N5_T2019_TT 2977 INT
N5_T2036_LACTOSE 2938.00 BOOL  ; LACTOSE PAA TANK
N5_T2036_LACTOSETEMP_HOEY 2938.01 BOOL  ; LACTOSE PAA TANK TEMP FOR HOEY
N5_T2036_LACTOSE_TID_OK 2938.05 BOOL  ; VALGT TID AVSLUTTET
N5_T2036_MANUELL_AAPNING 2936.00 BOOL
N5_T2036_SPERR 2902.00 BOOL
N5_T2037_LACTOSE 2938.02 BOOL  ; LACTOSE PAA TANK
N5_T2037_LACTOSETEMP_HOEY 2938.03 BOOL  ; LACTOSE PAA TANK TEMP FOR HOEY
N5_T2037_LACTOSE_TID_OK 2938.06 BOOL  ; VALGT TID AVSLUTTET
N5_T2037_SPERR 2902.01 BOOL
N5_T20_36_MAN 2936.00 BOOL
N5_T20_37_MAN 2936.01 BOOL
N5_V0640_INN 2923.00 BOOL
N5_V0641_INN 2923.01 BOOL
N5_V0642_INN 2923.02 BOOL
N5_V0643_INN 2923.03 BOOL
N5_V2001_UT 2923.08 BOOL
N5_V2002__UT 2923.09 BOOL
N5_V2003_UT 2923.10 BOOL
N5_V2004_UT 2923.11 BOOL
N5_V2005_UT 2923.12 BOOL
N5_V3742_UT 2906.00 BOOL
N5_V4250_INN 2940.11 BOOL
N5_V4251_INN 2940.12 BOOL
N5_V4255_INN 2940.13 BOOL
N5_V4305_INN 2917.07 BOOL  ; Z
N5_V8007_UT 2980.02 BOOL
N5_V8008_UT_N 2980.03 BOOL
N5_V80K4_KL_TRINN 2928 WORD
N5_VST60_K2_KL_AVSL 2921.12 BOOL
N5_VST80_K4_C25_KL_SLUTT 2900.14 BOOL
N5_VST90_K1_KLAPRING 2905.10 BOOL
N5_VST90_K1_TR07_TID_S 2956.03 BOOL  ; KURS 1 TRINN 07TID
N5_VST90_K1_TR21_TID_S 2956.04 BOOL  ; KURS 1 TRINN 21 TID
N5_VST90_K2_KLAPRING 2905.11 BOOL  ; KLAPRING AKTIV
N5_VST90_K2_TURSTOPP 2957.02 BOOL  ; STANSER TURPUMPENE.
N5_VST90_K3_KLAPRING 2905.12 BOOL  ; KLAPRING AKTIV
N5_VST90_K3_TR07_TID_S 2958.03 BOOL  ; KURS 3 TRINN 07TID
N6_0644_INN 3017.11 BOOL
N6_C21_DREN_STARTET 3002.00 BOOL
N6_C21_DREN_UTFOERT 3002.01 BOOL
N6_C21_STARTET 3002.02 BOOL
N6_C21_UTFOERT 3002.03 BOOL
N6_HL_T2028 3010.02 BOOL
N6_HL_T2029 3010.04 BOOL
N6_HL_T61_VST61 3020.00 BOOL
N6_HL_T62_VST60 3020.01 BOOL
N6_HL_T63_VST60 3020.02 BOOL
N6_HL_T64_VST60 3020.03 BOOL
N6_LL_T2028 3010.01 BOOL
N6_LL_T2029 3010.03 BOOL
N6_LUT_SOUPRANO 3040.00 BOOL
N6_P1060_AUTO 3001.00 BOOL  ; STYRER P2160_AUT0 FRA NODE6
N6_P2901_INN 3038.01 BOOL
N6_P2902_INN 3038.00 BOOL
N6_PGM515_C21_LINJETOEM 3002.04 BOOL  ; BENYTTES TIL AA TOEMME C21 LINJE
N6_PGM515_C46_LINJETOEM 3001.04 BOOL  ; BENYTTES TIL AA TOEMME C46 LINJE I N4 OG N5
N6_PGM552_KOE_DR 3053.06 BOOL
N6_PGM553_KOE_DR 3053.07 BOOL
N6_PGM554_KOE_DR 3053.08 BOOL
N6_PGM555_KOE_DR 3053.09 BOOL
N6_PGM556_KOE_DR 3053.10 BOOL
N6_R2801_INN 3038.02 BOOL
N6_R2901_INN 3038.03 BOOL
N6_RV_2017_INN 3010.00 BOOL
N6_SYRE_SOUPRANO 3040.01 BOOL
N6_TT_T2028 3011 CHANNEL
N6_V2801_INN 3015.00 BOOL
N6_V2802_INN 3015.01 BOOL
N6_V2803_INN 3015.02 BOOL
N6_V2804_INN 3015.03 BOOL
N6_V2805_INN 3015.04 BOOL
N6_V2806_INN 3015.05 BOOL
N6_V2807_INN 3015.06 BOOL
N6_V2810_INN 3015.07 BOOL
N6_V2811_INN 3015.08 BOOL
N6_V2820_INN 3015.09 BOOL
N6_V2830_INN 3015.10 BOOL
N6_V2860_INN 3015.11 BOOL
N6_V2901_INN 3016.00 BOOL
N6_V2902_INN 3016.01 BOOL
N6_V2903_INN 3016.02 BOOL
N6_V2904_INN 3016.03 BOOL
N6_V2905_INN 3016.04 BOOL
N6_V2906_INN 3016.05 BOOL
N6_V2907_INN 3016.06 BOOL
N6_V2908_INN 3016.07 BOOL
N6_V2909_INN 3017.10 BOOL
N6_V2910_INN 3016.08 BOOL
N6_V2912_1_INN 3016.09 BOOL
N6_V2913_1_INN 3016.11 BOOL
N6_V2920_INN 3016.13 BOOL
N6_V2922_1_INN 3016.14 BOOL
N6_V2923_1_INN 3017.00 BOOL
N6_V2930_INN 3017.02 BOOL
N6_V2931_INN 3017.03 BOOL
N6_V2941_INN 3017.04 BOOL
N6_V2942_INN 3017.05 BOOL
N6_V2948_INN 3017.06 BOOL
N6_V2960_INN 3017.07 BOOL
N6_V5504_INN 3000.00 BOOL
N6_V5506_INN 3000.01 BOOL
N6_V5604_INN 3000.02 BOOL
N6_V5606_INN 3000.03 BOOL
N6_V5704_INN 3000.04 BOOL
N6_V5706_INN 3000.05 BOOL
N6_V5804_INN 3000.06 BOOL
N6_V5806_INN 3000.07 BOOL
N6_V5904_INN 3000.08 BOOL
N6_V5906_INN 3000.09 BOOL
N6_V5911_INN 3000.10 BOOL
N6_V5921_INN 3000.11 BOOL
N6_V5922_INN 3000.12 BOOL
N6_VST60_K1_ER_KLAPRETRINN 3060 INT
N6_VST60_K1_KLAPRING 3006.05 BOOL
N6_VST60_K2_ER_KLAPRETRINN 3061 INT
N6_VSTE_N_STOPP 3020.05 BOOL
NETTV_TIL_VST80_MAN 1400.00 BOOL  ; NETTVANN TIL T81-84. OVERSTYRER NIVAA
NIVAA_T06_PR2 5140 UINT
NODE21_TELLER D1001 INT
NODE22_TELLER D1002 INT
NODE23_TELLER D1003 INT
NODE24_TELLER D1004 INT
NODE25_TELLER D1005 INT
NODE26_TELLER D1006 INT
NODE27_TELLER D1007 INT
NODE28_TELLER_1 D1008 INT
NODE29_TELLER_1 D1009 INT
NODE5_V_4302_INN 2935.04 BOOL
NODETELLERE_HJ D1010 INT
NODEVALG_1_GRAFIKK D3900 INT
NODEVALG_1_GRAFIKK_HJ D3901 INT
NODEVALG_2_GRAFIKK D3902 INT
NODEVALG_2_GRAFIKK_HJ D3903 INT
NODEVALG_3_GRAFIKK D3904 INT
NODEVALG_3_GRAFIKK_HJ D3905 INT
NODEVALG_4_GRAFIKK D3906 INT
NODEVALG_4_GRAFIKK_HJ D3907 INT
NODEVALG_5_GRAFIKK D3908 INT
NODEVALG_5_GRAFIKK_HJ D3909 INT
NODEVALG_6_GRAFIKK D3910 INT
NODEVALG_6_GRAFIKK_HJ D3911 INT
NODEVALG_7_GRAFIKK D3912 INT
NODEVALG_7_GRAFIKK_HJ D3913 INT
NODEVALG_8_GRAFIKK D3914 INT
NODEVALG_8_GRAFIKK_HJ D3915 INT
NODEVALG_9_GRAFIKK D3916 INT
NODEVALG_9_GRAFIKK_HJ D3917 INT
NOEDDOSERING_T84_INN 2701.02 BOOL  ; Z
NOEDDOSERING_T84_LAMP 2401.02 BOOL  ; LAMPE NOEDDOSERING
ON CF113 BOOL
ORD1 1991 CHANNEL
ORD2 1992 CHANNEL
P0101HZ1 D1440 CHANNEL  ; Z
P0101_AUTO 1054.07 BOOL
P0101_AUTOPAADRAG D20692 UINT
P0101_D D20653 CHANNEL
P0101_D_MEM D25063 CHANNEL
P0101_ER_FLOW D6124 WORD
P0101_ER_MENGDE D2012 WORD  ; ER VERDI I AKTUELL FUNKSJON
P0101_HAST_UT D20698 INT
P0101_HJ_TOT_MENGDE D2008 WORD
P0101_I D20652 CHANNEL
P0101_INN 2701.07 BOOL  ; Z
P0101_INN_FORS_S T0082 BOOL
P0101_INN_FORS_T 082 NUMBER
P0101_I_MEM D25062 CHANNEL
P0101_MAN 1004.07 BOOL
P0101_MAN_AUTO 1000.14 BOOL
P0101_MAN_HAST D6206 WORD
P0101_P D20651 CHANNEL
P0101_PROD_START 700.15 BOOL
P0101_PRS_FLOW D6200 WORD
P0101_P_MEM D25061 CHANNEL
P0101_REGN1 D20694 REAL
P0101_REGN2 D20696 REAL
P0101_RESET_REG D20650 CHANNEL
P0101_START_MENGDE D2022 WORD
P0101_TOT_MENGDE D2010 WORD
P0101_UT 2401.07 BOOL  ; Z
P0101_UT_FORS_S T0083 BOOL
P0101_UT_FORS_T 083 NUMBER
P0102_AUTO 1054.11 BOOL
P0102_INN 2700.10 BOOL  ; ISVANSPUMPE FOR L1.1 OG L1.2
P0102_MAN 1004.11 BOOL
P0102_UT 2400.10 BOOL  ; ISVANSPUMPE FOR L1.1 OG L1.2
P0111HZ1 D1442 CHANNEL  ; Z
P0111UT_FORS_T 088 NUMBER
P0111_AUTO 1054.08 BOOL
P0111_AUTOPAADRAG D20742 UINT
P0111_D D20703 CHANNEL
P0111_D_MEM D25073 CHANNEL
P0111_ER_FLOW D6128 WORD
P0111_ER_MENGDE D2112 WORD  ; ER VERDI I AKTUELL FUNKSJON
P0111_HAST_UT D20748 INT
P0111_HJ_TOT_MENGDE D2108 WORD
P0111_I D20702 CHANNEL
P0111_INN 2701.08 BOOL  ; Z
P0111_INN_FORS_S T0087 BOOL
P0111_INN_FORS_T 087 NUMBER
P0111_I_MEM D25072 CHANNEL
P0111_MAN 1004.08 BOOL
P0111_MAN_AUTO 1000.15 BOOL
P0111_MAN_HAST D6216 WORD
P0111_P D20701 CHANNEL
P0111_PROD_START 702.15 BOOL
P0111_PRS_FLOW D6210 WORD
P0111_P_MEM D25071 CHANNEL
P0111_REGN1 D20744 REAL
P0111_REGN2 D20746 REAL
P0111_RESET_REG D20700 CHANNEL
P0111_START_MENGDE D2122 WORD
P0111_TOT_MENGDE D2110 WORD
P0111_UT 2401.08 BOOL  ; Z
P0111_UT_FORS_S T0088 BOOL
P0201HZ1 D1444 CHANNEL  ; Z
P0201_AUTO 1054.09 BOOL
P0201_AUTOPAADRAG D20792 UINT
P0201_D D20753 CHANNEL
P0201_D_MEM D25083 CHANNEL
P0201_ER_FLOW D6132 WORD
P0201_ER_MENGDE D2212 WORD  ; ER VERDI I AKTUELL FUNKSJON
P0201_HAST_UT D20798 INT
P0201_HJ_TOT_MENGDE D2208 WORD
P0201_I D20752 CHANNEL
P0201_INN 2701.09 BOOL  ; Z
P0201_INNT_FORS_T 092 NUMBER
P0201_INN_FORS_S T0092 BOOL
P0201_I_MEM D25082 CHANNEL
P0201_MAN 1004.09 BOOL
P0201_MAN_AUTO 1001.00 BOOL
P0201_MAN_HAST D6226 WORD
P0201_P D20751 CHANNEL
P0201_PROD_START 704.15 BOOL
P0201_PRS_FLOW D6220 WORD
P0201_P_MEM D25081 CHANNEL
P0201_REGN1 D20794 REAL
P0201_REGN2 D20796 REAL
P0201_RESET_REG D20750 CHANNEL
P0201_START_MENGDE D2222 WORD
P0201_TOT_MENGDE D2210 WORD
P0201_UT 2401.09 BOOL  ; Z
P0201_UT_FORS_S T0093 BOOL
P0201_UT_FORS_T 093 NUMBER
P0202_AUTO 1054.12 BOOL
P0202_INN 2700.11 BOOL  ; ISVANSPUMPE FOR L2.1 OG L2.2
P0202_MAN 1004.12 BOOL
P0202_UT 2400.11 BOOL  ; ISVANSPUMPE FOR L2.1 OG L2.2
P0211HZ1 D1446 CHANNEL  ; Z
P0211_AUTO 1054.10 BOOL
P0211_AUTOPAADRAG D20842 UINT
P0211_D_MEM D25093 CHANNEL
P0211_ER_FLOW D6136 WORD
P0211_ER_MENGDE D2312 WORD  ; ER VERDI I AKTUELL FUNKSJON
P0211_HAST_UT D20848 INT
P0211_HJ_TOT_MENGDE D2308 WORD
P0211_I D20802 CHANNEL
P0211_INN 2701.10 BOOL  ; Z
P0211_INN_FORS_S T0097 BOOL
P0211_INN_FORS_T 097 NUMBER
P0211_I_MEM D25092 CHANNEL
P0211_MAN 1004.10 BOOL
P0211_MAN_AUTO 1001.01 BOOL
P0211_MAN_HAST D6236 WORD
P0211_P D20801 CHANNEL
P0211_PROD_START 706.15 BOOL
P0211_PRS_FLOW D6230 WORD
P0211_P_MEM D25091 CHANNEL
P0211_REGN1 D20844 REAL
P0211_REGN2 D20846 REAL
P0211_RESET_REG D20800 CHANNEL
P0211_START_MENGDE D2322 WORD
P0211_TOT_MENGDE D2310 WORD
P0211_UT 2401.10 BOOL  ; Z
P0211_UT_FORS_S T0098 BOOL
P0211_UT_FORS_T 098 NUMBER
P0351_AUTO 1054.00 BOOL
P0351_INN 2701.13 BOOL  ; Z
P0351_MAN 1004.00 BOOL
P0351_UT 2401.13 BOOL  ; Z
P0361_AUTO 1054.01 BOOL
P0361_INN 2701.14 BOOL  ; Z
P0361_MAN 1004.01 BOOL
P0361_UT 2401.14 BOOL  ; Z
P0501_AUTO 1054.06 BOOL
P0501_INN 2701.12 BOOL  ; Z
P0501_MAN 1004.06 BOOL
P0501_UT 2401.12 BOOL  ; Z
P1060_AUTO 1056.14 BOOL
P1060_INN 2704.04 BOOL  ; ISVANN GALLERI
P1060_MAN 1006.14 BOOL
P1060_UT 2404.04 BOOL  ; ISVANN GALLERI
P1101 OPPSKALERING
P1101_INN_N5 2803.02 BOOL
P1102_INN_N5 2803.03 BOOL
P1940_I_DR_N5 2803.01 BOOL  ; UHT AVD. INNG. DRIFT
P2021_I_DR_N5 2819.05 BOOL  ; UHT AVD. INNG. DRIFT
P2025_I_DRK_PR2 5112.03 BOOL  ; UHT AVD. INNG.  DRIFTSKLAR
P2028_INN_N5 2819.07 BOOL  ; UHT AVD. INNG. DRIFT
P2028_SIST_FRA_2036 2905.01 BOOL
P2028_SIST_FRA_2037 2905.05 BOOL
P2028_UT_N5 2919.13 BOOL  ; UHT AVD
P2029_INN_N5 2819.08 BOOL  ; UHT AVD. INNG. DRIFT
P2029_SIST_FRA_2036 2905.02 BOOL
P2029_SIST_FRA_2037 2905.06 BOOL
P2029_UT_N5 2919.15 BOOL  ; UHT AVD
P2031_SIST_FRA_2036 2905.00 BOOL
P2031_SIST_FRA_2037 2905.04 BOOL
P2039_INN_N5 2821.02 BOOL
P2044_SIST_FRA_2036 2905.03 BOOL
P2044_SIST_FRA_2037 2905.07 BOOL
P2060_INN 2704.03 BOOL  ; ISVANN UHT
P2060_UT 2404.03 BOOL  ; ISVANN UHT
P2101 BRA_PID
P2101_AUTO 1056.04 BOOL
P2101_D D21053 CHANNEL
P2101_FETT_FLOETE_KG D6178 REAL
P2101_FLOETE_FETTPR D6170 REAL
P2101_HJ_FETT_FLOETE_KG D7852 REAL  ; RESULTAT FOER KORRIGERING VHA EGENVEKT
P2101_HJ_FLOETE_FETTPR D7854 REAL  ; FLOETE FETTPROSENT DIV PAA 100
P2101_HJ_MELK_DIF_FETT_INN_UT D7850 REAL  ; DIFFERANSE FETT% INN OG UT/100
P2101_HJ_PRS_MELK_INN D7856 REAL  ; MELK TIL PAST. I 0-1000 1000=20000L/T
P2101_I D21052 CHANNEL
P2101_INN 2700.12 BOOL
P2101_MAN 1006.04 BOOL
P2101_MAN_AUTO 1001.06 BOOL
P2101_MELK_DIF_FETT_INN_UT D6172 REAL  ; DIFFERANSE FETT% INN OG UT
P2101_MELK_FETTPR_INN D6166 REAL
P2101_MELK_FETTPR_UT D6168 REAL
P2101_MELK_INN D6174 REAL  ; MELK TIL PAST. I L/T
P2101_MELK_TIL_FLOETE D6180 REAL  ; MELKEMENGDE TIL FLOETELOEP I L/T
P2101_MELK_UT D6176 REAL  ; UT AV PAST. I L/T
P2101_OPPSKALER OPPSKALERING
P2101_P D21051 CHANNEL
P2101_PAADRAG D1492 UINT
P2101_PAADRAG_FLT D22100 REAL
P2101_PRS D3116 WORD
P2101_PRS_FRYS D3170 WORD
P2101_PRS_L_PR_T D4172 WORD  ; 0-20000
P2101_PRS_MAN D3118 WORD
P2101_PRS_MELK_INN D6162 WORD  ; MELK TIL PAST. I 0-1000 1000=20000L/T
P2101_PRS_REEL D3162 WORD  ; 0-20000L/T
P2101_UT 2400.12 BOOL
P2102_AUTO 1056.05 BOOL
P2102_INN 2700.14 BOOL
P2102_MAN 1006.05 BOOL
P2102_UT 2400.14 BOOL
P2103HZ1 D1490 UINT
P2103_AUTO 1055.07 BOOL  ; FORELOEPIG BARE ON/OFF STYRING. MULIGHET OGSAA AA STYRE PID MED 1=AUTOVERDI, 0=MANVERDI.
P2103_AUTOPAADRAG D20310 UINT
P2103_D_MEM D25143 UINT
P2103_INN 2701.03 BOOL
P2103_I_MEM D25142 UINT
P2103_MAN 1005.07 BOOL
P2103_OPPSKALER OPPSKALERING
P2103_PAADRAG D20316 UINT
P2103_PRESET D20300 UINT
P2103_PRS D8891 UINT
P2103_PRS_FRYS D3172 WORD
P2103_P_MEM D25141 UINT
P2103_TEMP1 D42 UDINT
P2103_TEMP2 D46 UDINT
P2103_UT 2401.03 BOOL
P2104_AUTO 1056.06 BOOL
P2104_D D22003 CHANNEL
P2104_FAKTOR_REAL D22132 REAL
P2104_I D22002 CHANNEL
P2104_INN 2700.13 BOOL
P2104_MAN 1006.06 BOOL
P2104_MAN_AUTO 1001.07 BOOL
P2104_OPPSKALER OPPSKALERING
P2104_P D22001 CHANNEL
P2104_PAADRAG D1494 UINT
P2104_PAADRAG_FAKT D22106 REAL
P2104_PAADRAG_FAKT_REAL D22104 REAL
P2104_PROSENT_INT D21118 INT
P2104_PROSENT_REAL D22130 REAL
P2104_PRS D3122 WORD
P2104_PRS_MAN D3124 WORD
P2104_REGN1 D22044 REAL
P2104_REGN2 D22046 REAL
P2104_UT 2400.13 BOOL
P2160_AUTO 1056.12 BOOL  ; ISVANN SKUMMESAL
P2160_INN 2704.02 BOOL  ; ISVANN SKUMMESAL
P2160_MAN 1006.12 BOOL
P2160_UT 2404.02 BOOL  ; ISVANN SKUMMESAL
P21_BLK_TOM_MELK_INN 4502.04 BOOL  ; BLK TOM MELK INN
P21_Betinget_Omslag_DP2 226.00 BOOL
P21_DP1_DIFF_TRYKK D3604 INT  ; B2102 - B2101
P21_DP1_OK 4803.00 BOOL  ; TRYKK  DP1 OK
P21_DP1_OK_UTFORS_S T0803 BOOL
P21_DP1_OK_UTFORS_T 0803 NUMBER
P21_DP1_OMSLAG 4803.05 BOOL  ; TRYKKOMSLAG DP1
P21_DP1_SPERR_OMSLAG 4803.09 BOOL  ; TRYKKOMSLAG DP1 SPERRET
P21_DP2_DIFF_TRYKK D3606 INT  ; B2104 - B2103
P21_DP2_OK 4803.01 BOOL  ; TRYKK  DP2 OK
P21_DP2_OK_UTFORS_S T0804 BOOL
P21_DP2_OMSLAG 4803.06 BOOL  ; TRYKKOMSLAG DP2
P21_DP2_Omslagsteller 220 INT
P21_DP2_SPERR_OMSLAG 4803.10 BOOL  ; TRYKKOMSLAG DP2 SPERRET
P21_DREN_FOERST_TIL_GR08 4802.07 BOOL
P21_ER_MELK_INN D3626 DINT
P21_ER_MELK_INN_ER_S_TID D3632 INT  ; SIKKERHETSTID VED FYLLING AV MELK
P21_ER_MELK_INN_PRS_S_TID D3630 INT  ; SIKKERHETSTID VED FYLLING AV MELK
P21_ER_MELK_INN_ST_MENGDE D3628 DINT  ; Q21 VERDI VED START
P21_ER_MENGDE_INN D3602 DINT  ; MENGDE I LITER
P21_ER_VANN_INN D3642 DINT  ; ¨
P21_FEIL_S T0808 BOOL
P21_FEIL_T 0808 NUMBER
P21_FLOW_OK 4803.02 BOOL  ; FLOW OK
P21_FLOW_OMSLAG 4803.07 BOOL  ; FOR HOEY FLOW
P21_FLOW_SPERR_OMSLAG 4803.11 BOOL  ; FOR HOEY FLOW SPERRET
P21_HEV_MOTTRYKK 226.06 BOOL
P21_HJ_TOT_MENGDE D3618 DINT  ; MENGDE I LITER
P21_ISV_DIFF_TRYKK D3736 INT
P21_ISV_KONTROLL 4801.12 BOOL
P21_MELK_INN 4502.05 BOOL  ; BLK TOM MELK INN
P21_MELK_INN_ER_MENGDE D3646 DINT
P21_MELK_INN_S T0828 BOOL  ; BLK TOM
P21_MELK_INN_ST_MENGDE D3648 DINT  ; Q21 VERDI VED START
P21_MELK_INN_T 0828 NUMBER  ; BLK TOM
P21_MELK_LAGER_N5 2800.02 BOOL
P21_MELK_T2009_N5 2800.01 BOOL
P21_MELK_TIL_ANL_DRIFT 4802.04 BOOL  ; DRIFSIGNAL TIL Q21
P21_MELK_TIL_ANL_RESET 4802.05 BOOL  ; RESETSIGNAL TIL Q21
P21_MELK_VED_T2009 4802.00 BOOL
P21_MELK_VED_TGR08 4802.02 BOOL
P21_MELK_VED_TGR08_N6 2821.12 BOOL
P21_MELK_VED_TGR09 4802.03 BOOL
P21_MELK_VED_TGR09_N6 2807.00 BOOL
P21_MELK_VED_UHT 4802.01 BOOL
P21_PAST_TEMP_OK 4803.03 BOOL  ; PASTEURISERINGSTEMP OK
P21_PRS_MENGDE_INN D3600 DINT  ; MENGDE I LITER
P21_SKRIVER_UT 1820.00 BOOL
P21_SKUDDPAUSE_S T0810 BOOL
P21_SKUDDPAUSE_T 0810 NUMBER
P21_STOPPTID_S T0809 BOOL
P21_STOPPTID_T 0809 NUMBER
P21_TEMP_OMSLAG 4803.08 BOOL  ; FOR LAV TEMPERATUR
P21_TEMP_SPERR_OMSLAG 4803.12 BOOL  ; FOR LAV TEMPERATUR SPERRET
P21_TILLEGG_MOTTRYKK 231 INT
P21_TOT_MENGDE_GR08 D3608 DINT  ; MENGDE I LITER
P21_TOT_MENGDE_GR09 D3610 DINT  ; MENGDE I LITER
P21_TOT_MENGDE_RETUR D3614 DINT  ; MENGDE I LITER
P21_TOT_MENGDE_UHT D3612 DINT  ; MENGDE I LITER
P21_UT_FORS_TELLERR_S T0807 BOOL  ; PAST21  TIL T.GR08 OG 09
P21_UT_FORS_TELLERR_T 0807 NUMBER  ; PAST21  TIL T.GR08 OG 09
P21_UT_I_LINJE 4802.10 BOOL  ; UT PAA LINJER TIL TANKER
P21_UT_I_LINJE_N5 2802.09 BOOL
P21_UT_TEMP_OK 4803.04 BOOL  ; UT-TEMP AV PAST OK
P21_VANN_INN_AVSL 4502.06 BOOL  ; BLK TOM VANN INN VED AVSLUTNING
P21_VANN_INN_ST_MENGDE D3644 DINT  ; Q21 VERDI VED START
P21_VANN_I_LINJE 4802.08 BOOL
P21_VASKER_AVBRUDD_S T0820 BOOL
P21_VASKER_AVBRUDD_T 0819 NUMBER
P2201 BRA_PID
P2201_AUTO 1056.07 BOOL
P2201_D D23003 CHANNEL
P2201_FETT_FLOETE_KG D6278 REAL
P2201_FLOETE_FETTPR D6270 REAL
P2201_HJ_D1496 D3228 WORD
P2201_HJ_FETT_FLOETE_KG D7952 REAL  ; RESULTAT FOER KORRIGERING VHA EGENVEKT
P2201_HJ_FLOETE_FETTPR D7954 REAL  ; FLOETE FETTPROSENT DIV PAA 100
P2201_HJ_MELK_DIF_FETT_INN_UT D7950 REAL  ; DIFFERANSE FETT% INN OG UT/100
P2201_HJ_PRS_MELK_INN D7956 REAL  ; MELK TIL PAST. I 0-1000 1000=20000L/T
P2201_I D23002 CHANNEL
P2201_INN 2701.00 BOOL  ; Z
P2201_MAN 1006.07 BOOL
P2201_MAN_AUTO 1001.09 BOOL
P2201_MAN_PRS D3218 WORD  ; 0-1000
P2201_MELK_DIF_FETT_INN_UT D6272 REAL  ; DIFFERANSE FETT% INN OG UT
P2201_MELK_FETTPR_INN D6266 REAL
P2201_MELK_FETTPR_UT D6268 REAL
P2201_MELK_INN D6274 REAL  ; MELK TIL PAST. I L/T
P2201_MELK_TIL_FLOETE D6280 REAL  ; MELKEMENGDE TIL FLOETELOEP I L/T
P2201_MELK_UT D6276 REAL  ; UT AV PAST. I L/T
P2201_OPPSKALER OPPSKALERING
P2201_P D23001 CHANNEL
P2201_PAADRAG D1496 UINT
P2201_PAADRAG_FLT D22110 REAL
P2201_PRS D3216 WORD  ; 0-1000
P2201_PRS_L_PR_T D4272 WORD  ; 0-20000
P2201_PRS_MELK_INN D6262 WORD  ; MELK TIL PAST. I 0-1000 1000=20000L/T
P2201_UT 2401.00 BOOL  ; Z
P2202_AUTO 1056.08 BOOL
P2202_INN 2701.04 BOOL  ; Z
P2202_MAN 1006.08 BOOL
P2202_UT 2401.04 BOOL  ; Z
P2203_AUTO 1056.10 BOOL
P2203_INN 2701.05 BOOL  ; Z
P2203_MAN 1006.10 BOOL
P2203_UT 2401.05 BOOL  ; Z
P2204_AUTO 1056.09 BOOL
P2204_D D23023 CHANNEL
P2204_FAKTOR_REAL D22122 REAL
P2204_I D23022 CHANNEL
P2204_INN 2701.06 BOOL  ; Z
P2204_MAN 1006.09 BOOL
P2204_MAN_AUTO 1001.11 BOOL
P2204_MAN_PRS D3232 WORD  ; 0-1000
P2204_MELK 4812.00 BOOL
P2204_OPPSKALER OPPSKALERING
P2204_P D23021 CHANNEL
P2204_PAADRAG D1498 UINT
P2204_PAADRAG_FAKT D22116 INT
P2204_PAADRAG_FAKT_REAL D22112 REAL
P2204_PROSENT_INT D22118 INT
P2204_PROSENT_REAL D22120 REAL
P2204_PRS D3230 WORD  ; 0-1000
P2204_UT 2401.06 BOOL  ; Z
P22_BLK_TOM_MELK_INN 4512.04 BOOL  ; BLK TOM MELK INN
P22_Betinget_Omslag_DP2 216.00 BOOL
P22_C25_VASKET_DREN_T T0906 BOOL
P22_DP1_DIFF_TRYKK D3704 INT  ; B2202 - B2201
P22_DP1_OK 4813.00 BOOL  ; TRYKK  DP1 OK
P22_DP1_OK_UTFORS_S T0805 BOOL
P22_DP1_OK_UTFORS_T 0805 NUMBER
P22_DP1_OMSLAG 4813.05 BOOL  ; TRYKKOMSLAG DP1
P22_DP1_SPERR_OMSLAG 4813.09 BOOL  ; TRYKKOMSLAG DP1 SPERRET
P22_DP2_DIFF_TRYKK D3706 INT  ; B2204¨ - B2203
P22_DP2_OK 4813.01 BOOL  ; TRYKK  DP2 OK
P22_DP2_OK_UTFORS_S T0806 BOOL
P22_DP2_OK_UTFORS_T 0806 NUMBER
P22_DP2_OMSLAG 4813.06 BOOL  ; TRYKKOMSLAG DP2
P22_DP2_Omslagsteller 220 INT
P22_DP2_SPERR_OMSLAG 4813.10 BOOL  ; TRYKKOMSLAG DP2  SPERRET
P22_DP3_DIFF_TRYKK D3718 INT
P22_DP3_OK 4814.07 BOOL
P22_DP3_OK_UTFORS_S T0843 BOOL
P22_DP3_OMSLAG 4814.03 BOOL  ; TRYKKOMSLAG DP1
P22_DP3_SPERR_OMSLAG 4814.13 BOOL  ; TRYKKOMSLAG DP1 SPERRET
P22_DREN_FOERST_TIL_GR08 4812.07 BOOL
P22_ER_MELK_INN D3726 DINT
P22_ER_MELK_INN_ER_S_TID D3732 INT  ; SIKKERHETSTID VED FYLLING AV MELK
P22_ER_MELK_INN_PRS_S_TID D3730 INT  ; SIKKERHETSTID VED FYLLING AV MELK
P22_ER_MELK_INN_ST_MENGDE D3728 DINT  ; Q22 VERDI VED START
P22_ER_MENGDE_INN D3702 DINT  ; '
P22_ER_VANN_INN D3762 DINT  ; ¨
P22_FEIL_T 0813 NUMBER
P22_FLOW_OK 4813.02 BOOL  ; FLOW OK
P22_FLOW_OMSLAG 4813.07 BOOL  ; FOR HOEY FLOW
P22_FLOW_SPERR_OMSLAG 4813.11 BOOL  ; FOR HOEY FLOW SPERRET
P22_FLOW_SPERR_S T0817 BOOL
P22_FLOW_SPERR_T 0817 NUMBER
P22_GR08_FORS_C_RESET_S T0811 BOOL  ; PAST22  TIL T.GR08
P22_GR08_FORS_C_RESET_T 0811 NUMBER  ; PAST22  TIL T.GR08
P22_GR09_FORS_C_RESET_S T0812 BOOL  ; PAST22  TIL T.GR09
P22_GR09_FORS_C_RESET_T 0812 NUMBER  ; PAST22  TIL T.GR09
P22_HCELLE_OML 924.00 BOOL
P22_HC_FLOW_AV_S T0819 BOOL
P22_HC_FLOW_AV_T 0820 NUMBER
P22_HC_TMU_S T0818 BOOL
P22_HC_TMU_T 0818 NUMBER
P22_HJ_TOT_MENGDE D3718 DINT  ; MENGDE I LITER
P22_ISV_DIFF_TRYKK D3734 INT
P22_ISV_KONTROLL 4811.12 BOOL
P22_MELK_INN 4512.05 BOOL  ; BLK TOM MELK INN
P22_MELK_INN_ER_MENGDE D3766 DINT
P22_MELK_INN_S T0832 BOOL  ; BLK TOM
P22_MELK_INN_ST_MENGDE D3768 DINT  ; Q22 VERDI VED START
P22_MELK_INN_T 0832 NUMBER  ; BLK TOM
P22_MELK_LAGER_N5 2800.03 BOOL
P22_MELK_TIL_ANL_DRIFT 4812.04 BOOL  ; DRIFSIGNAL TIL Q22
P22_MELK_TIL_ANL_RESET 4812.05 BOOL  ; RESETSIGNAL TIL Q22
P22_MELK_VED_GR08 2829.00 BOOL
P22_MELK_VED_TGR08 4812.02 BOOL
P22_MELK_VED_TGR09 4812.03 BOOL
P22_MELK_VED_TGR09_N6 2807.01 BOOL
P22_MELK_VED_UHT 4812.01 BOOL
P22_PAST_TEMP_OK 4813.03 BOOL  ; PASTEURISERINGSTEMP OK
P22_PRS_MENGDE_INN D3700 DINT  ; '
P22_RESET_TOT_MENGDE_UT 4811.11 BOOL
P22_SKRIVER_UT 1820.01 BOOL
P22_STOPPTID_T 0814 NUMBER
P22_SURT_UT_20GR 4814.08 BOOL
P22_TEMP_OMSLAG 4813.08 BOOL  ; FOR LAV TEMPERATUR
P22_TEMP_SPERR_OMSLAG 4813.12 BOOL  ; FOR LAV TEMPERATUR SPERRET
P22_TGR08_N6 2821.13 BOOL
P22_TOT_MENGDE_GR08 D3708 DINT  ; MENGDE I LITER
P22_TOT_MENGDE_GR09 D3710 DINT  ; MENGDE I LITER
P22_TOT_MENGDE_RETUR D3714 DINT  ; MENGDE I LITER
P22_TOT_MENGDE_UHT D3712 DINT  ; MENGDE I LITER
P22_UT_I_LINJE 4812.10 BOOL  ; UT PAA LINJER TIL TANKER
P22_UT_I_LINJE_N6 2802.10 BOOL
P22_UT_TEMP_OK 4813.04 BOOL  ; UT-TEMP AV PAST OK
P22_VANN_INN_AVSL 4512.06 BOOL  ; BLK TOM VANN INN VED AVSLUTNING
P22_VANN_INN_ST_MENGDE D3764 DINT  ; Q22 VERDI VED START
P22_VANN_I_LINJE 4812.08 BOOL
P22_VASKER_AVBRUDD_S T0821 BOOL
P22_VASKER_AVBRUDD_T 0821 NUMBER
P2301 BRA_PID
P2301PAADRAG D1500 UINT  ; 0-1000
P2301_AUTO 1056.02 BOOL
P2301_D D23043 UINT
P2301_ER_TID_MANVERDI D3356 WORD
P2301_I D23042 UINT
P2301_INN 2702.12 BOOL  ; Z
P2301_MAN 1006.02 BOOL
P2301_MAN_AUTO 1001.13 BOOL  ; MAN=1
P2301_MAN_PRS D3318 UINT  ; D3318
P2301_OPPSKALER OPPSKALERING
P2301_P D23041 UINT
P2301_PRS D3316 WORD  ; '
P2301_PRS_ENDRE_MAN_PRS 4820.08 BOOL
P2301_PRS_L_PR_T D4372 WORD  ; 0-8000
P2301_PRS_REEL D3352 UINT  ; 0-4000L/T
P2301_PRS_TID_MANVERDI D3354 WORD
P2301_UT 2402.12 BOOL  ; Z
P2302_AUTO 1056.03 BOOL
P2302_INN 2702.13 BOOL
P2302_MAN 1006.03 BOOL
P2302_UT 2402.13 BOOL  ; Z
P2304_ANALOG_UT OPPSKALERING
P2304_AUTO 1056.13 BOOL
P2304_CIP_SETP D3886 INT
P2304_INN 2703.02 BOOL
P2304_MAN 1006.13 BOOL
P2304_PAADRAG D1432 UINT
P2304_PROD_SETP D3887 INT
P2304_UT 2403.02 BOOL
P23_ACC_MENGDE_TIL_CONT D3850 DINT  ; MENGDE I LITER
P23_ACC_MENGDE_TIL_GR10 D3826 DINT  ; MENGDE I LITER
P23_ACC_MENGDE_TIL_T2009 D3834 DINT  ; MENGDE I LITER
P23_BLKNIV_RUNDL_S T0816 BOOL
P23_BLKNIV_RUNDL_T 0816 NUMBER
P23_C25_VASKET 4822.10 BOOL  ; BENYTTES TIL DREN AV VANN FRA T2009
P23_CONT_TOT_RESET 4820.11 BOOL
P23_DIFFTRYKK_SEKSJ_4 OPPSKALERING
P23_DIFF_TEMP D3898 DINT
P23_DIFF_TEMP_OK 4826.09 BOOL
P23_DIFF_TEMP_OMSLAG 4826.08 BOOL
P23_DIFTRYKK_SEKSJ2_OPPSKALERING OPPSKALERING
P23_DIFTRYKK_SEKSJ_3 OPPSKALERING
P23_DP1_DIFF_TRYKK D3890 DINT
P23_DP1_OK 4826.00 BOOL
P23_DP1_OMSLAG 4826.04 BOOL
P23_DP1_SPERR_OMSLAG 4815.00 BOOL
P23_DP2_DIFF_TRYKK D3892 DINT
P23_DP2_OK 4826.01 BOOL
P23_DP2_OMSLAG 4826.05 BOOL
P23_DP2_SPERR_OMSLAG 4815.01 BOOL
P23_DP3_DIFF_TRYKK D3894 DINT
P23_DP3_OK 4826.02 BOOL
P23_DP3_OMSLAG 4826.06 BOOL
P23_DP3_SPERR_OMSLAG 4815.02 BOOL
P23_DP4_DIFF_TRYKK D3896 DINT
P23_DP4_OK 4826.03 BOOL
P23_DP4_OMSLAG 4826.07 BOOL
P23_DP4_SPERR_OMSLAG 4815.03 BOOL
P23_ER_DRENSMENGDE D3878 DINT
P23_ER_FLOETE_I_ANLEGG D3846 DINT
P23_ER_MENGDE_INN D3802 DINT  ; MENGDE I LITER
P23_ER_MENGDE_TIL_UHT D3830 DINT  ; MENGDE I LITER
P23_ER_VANN_INN D3862 DINT  ; ¨
P23_FLOETE_INN_ER_MENGDE D3866 DINT
P23_FLOETE_INN_PRS_MENGDE D3872 DINT
P23_FLOETE_INN_ST_MENGDE D3868 DINT  ; Q23 VERDI VED START
P23_FLOETE_VED_TGR10_N6 2807.02 BOOL
P23_FLOW_OK 4823.02 BOOL  ; FLOW OK
P23_FLOW_OMSLAG 4823.07 BOOL  ; FOR HOEY FLOW
P23_FLOW_SPERR_OMSLAG 4823.11 BOOL  ; FOR HOEY FLOW SPERRET
P23_GR10_TOT_RESET 4820.10 BOOL
P23_IMP_FLOETE_I_ANLEGG 4522.02 BOOL
P23_ISV_KONTROLL 4821.12 BOOL
P23_MELK_INN 4522.05 BOOL  ; BLK TOM MELK INN
P23_PAST_TEMP_OK 4823.03 BOOL  ; PASTEURISERINGSTEMP OK
P23_PRS_DRENSMENGDE D3876 DINT
P23_PRS_FLOETE_I_ANLEGG D3844 DINT
P23_PRS_MENGDE_INN D3800 DINT  ; MENGDE I LITER
P23_PRS_MENGDE_TIL_CONT D3832 INT  ; MENGDE I LITER
P23_PRS_MENGDE_TIL_GR10 D3824 INT  ; MENGDE I LITER
P23_PRS_MENGDE_TIL_T2009 D3818 INT  ; MENGDE I LITER
P23_PRS_MENGDE_TIL_UHT D3828 INT  ; MENGDE I LITER
P23_PRS_VANN_INN D3870 DINT  ; ¨
P23_SKRIVER_UT 1820.02 BOOL
P23_START_FLOETE_I_ANLEGG D3848 DINT  ; STARTMENGDE
P23_T2009_TOT_RESET 4820.12 BOOL
P23_TEMP_OMSLAG 4823.08 BOOL  ; FOR LAV TEMPERATUR
P23_TEMP_SPERR_OMSLAG 4823.12 BOOL  ; FOR LAV TEMPERATUR SPERRET
P23_TOT_MENGDE_TIL_CONT D3842 DINT  ; MENGDE I LITER
P23_TOT_MENGDE_TIL_GR10 D3836 DINT  ; MENGDE I LITER
P23_TOT_MENGDE_TIL_GR10_RESET 4821.07 BOOL
P23_TOT_MENGDE_TIL_T2009 D3840 DINT  ; MENGDE I LITER
P23_TOT_MENGDE_TIL_T2009_RESET 4821.09 BOOL
P23_TOT_MENGDE_TIL_UHT D3838 DINT  ; MENGDE I LITER
P23_TOT_MENGDE_TIL_UHT_RESET 4821.08 BOOL
P23_UHT_TOT_RESET 4820.09 BOOL
P23_UT_TEMP_OK 4823.04 BOOL  ; UT-TEMP AV PAST OK
P23_VANN_INN_AVSL 4522.06 BOOL  ; BLK TOM VANN INN VED AVSLUTNING
P23_VANN_INN_ST_MENGDE D3864 DINT  ; Q23 VERDI VED START
P23_VASKER_AVBRUDD_S T0822 BOOL
P23_VASKER_AVBRUDD_T 0822 NUMBER
P2401_AUTO 1056.01 BOOL
P2401_INN 2702.14 BOOL
P2401_MAN 1006.01 BOOL
P2401_UT 2402.14 BOOL  ; Z
P2601_AUTO 1056.15 BOOL  ; MOTTAK OEKOMELK
P2601_INN 2704.01 BOOL  ; MOTTAK OEKOMELK
P2601_MAN 1006.15 BOOL  ; MOTTAK OEKOMELK
P2601_UT 2404.01 BOOL  ; MOTTAK OEKOMELK
P2901_UT_N6 2864.01 BOOL
P2902_UT_N6 2864.00 BOOL
P3201_AUTO 1055.04 BOOL
P3201_I 2702.04 BOOL
P3201_MAN 1005.04 BOOL
P3201_U 2402.04 BOOL
P3601_AUTO 1055.00 BOOL
P3601_INN 2702.02 BOOL
P3601_MAN 1005.00 BOOL
P3601_UT 2402.02 BOOL
P4401_AUTO 1055.15 BOOL
P4401_INN 2702.10 BOOL
P4401_MAN 1005.15 BOOL
P4401_UT 2402.10 BOOL
P4501_AUTO 1056.00 BOOL  ; ¨
P4501_INN 2702.11 BOOL
P4501_MAN 1006.00 BOOL
P4501_UT 2402.11 BOOL
P4501_VASK 748.00 BOOL
P6010_UT_N6 2864.04 BOOL
P6012_UT_N6 2864.06 BOOL
P6020_UT_N6 2864.05 BOOL
P8001INN D1666 REAL  ; Z
P8001_AUTO 1052.10 BOOL
P8001_D_MEM D25003 CHANNEL
P8001_INN 2700.00 BOOL  ; Z
P8001_I_MEM D25002 CHANNEL
P8001_MAN 1002.10 BOOL
P8001_PAADRAG_MAN D8644 INT
P8001_PRS D8642 UINT
P8001_P_MEM D25001 CHANNEL
P8001_UT 2400.00 BOOL  ; Z
P8002INN D1668 REAL  ; TEMP DYPVANNSUTSLIPP
P8002_AUTO 1052.11 BOOL
P8002_D_MEM D25023 CHANNEL
P8002_INN 2700.01 BOOL  ; Z
P8002_I_MEM D25022 CHANNEL
P8002_MAN 1002.11 BOOL
P8002_PAADRAG_MAN D8744 DWORD
P8002_PRS D8742 UINT
P8002_P_MEM D25021 CHANNEL
P8002_UT 2400.01 BOOL  ; Z
P8003INN D1670 REAL  ; Z
P8003_AUTO 1052.12 BOOL
P8003_D_MEM D25043 CHANNEL
P8003_INN 2700.02 BOOL  ; Z
P8003_I_MEM D25042 CHANNEL
P8003_MAN 1002.12 BOOL
P8003_PAADRAG_MAN D8844 CHANNEL
P8003_PRS D8842 UINT
P8003_P_MEM D25041 CHANNEL
P8003_UT 2400.02 BOOL  ; Z
P8004_AUTO 1053.14 BOOL
P8004_INN 2701.11 BOOL  ; Z
P8004_MAN 1003.14 BOOL
P8004_TID_STARTVENT T0442 BOOL  ; FORSINKER PUMPESTART
P8004_UT 2401.11 BOOL  ; Z
P8010_FEILFORSINK T0152 BOOL  ; FORSINKER FEILMELDING FRA  FREKVENSOMF.
P8010_PRS D8610 UINT
P8011_AUTO 1053.13 BOOL
P8011_INN 2700.03 BOOL  ; VST80-K1-TUR SIRK.PUMPE
P8011_INN_N 2700.06 BOOL  ; Z
P8011_MAN 1003.13 BOOL
P8011_UT 2400.03 BOOL  ; VST80-K1-TUR SIRK.PUMPE
P8011_UT_N 2400.06 BOOL  ; Z
P8012_AUTO 1054.02 BOOL
P8012_INN 2700.07 BOOL  ; Z
P8012_MAN 1004.02 BOOL
P8012_UT 2400.07 BOOL  ; Z
P8023_AUTO 1054.05 BOOL
P8023_INN 2508.13 BOOL  ; Z
P8023_MAN 1004.05 BOOL
P8023_UT 2208.13 BOOL  ; Z
P8024_AUTO 1057.02 BOOL
P8024_INN 2702.15 BOOL  ; Z
P8024_MAN 1007.02 BOOL
P8024_UT 2402.15 BOOL  ; Z
P8026_AUTO 1055.14 BOOL
P8026_INN 2702.09 BOOL
P8026_MAN 1005.14 BOOL
P8026_UT 2402.09 BOOL
P8030_AUTO 1054.03 BOOL
P8030_INN 2700.08 BOOL  ; Z
P8030_MAN 1004.03 BOOL
P8030_UT 2400.08 BOOL  ; Z
P8031_AUTO 1054.04 BOOL
P8031_INN 2700.09 BOOL  ; Z
P8031_MAN 1004.04 BOOL
P8031_UT 2400.09 BOOL  ; Z
P8222_AUTO 1053.01 BOOL
P8322_AUTO 1053.02 BOOL
P8422_AUTO 1053.03 BOOL
PAADRAG_MAN_V8024 D8602 CHANNEL
PAADRAG_MAN_V8024_MID D9602 CHANNEL  ; SKAL_FJERNES
PAADRAG_TIL_P8001 D1400 CHANNEL  ; VST80 TURPUMPE KURS1 HAST. TIL FR.OMF. P8010
PAADRAG_TIL_P8002 D1402 CHANNEL  ; VST80 TURPUMPE KURS2 HAST. TIL FR.OMF. P8002
PAADRAG_TIL_P8003 D1404 CHANNEL
PAADRAG_V8014 D20098 REAL
PAADRAG_V8024 D20198 INT
PAADRAG_V8034 D20298 INT
PAN27_C06_LAMPE 2100.00 BOOL
PAN27_C07_LAMPE 2100.01 BOOL
PAN27_C08_LAMPE 2100.02 BOOL
PANEL27_C06_START_TR 2603.01 BOOL
PANEL27_C06_STOPPER_TUR 1319.06 BOOL  ; STOPPER  TURPUMPE OG TIDSFORLOEP
PANEL27_C06_STOPP_TUR_IMP 1319.05 BOOL  ; IMPULS STOPP  TURPUMPE OG TIDSFORLOEP
PANEL27_C06_STOPP_TUR_TR 2603.11 BOOL
PANEL27_C07_START_TR 2603.02 BOOL
PANEL27_C08_START_TR 2603.03 BOOL  ; Panel 27_Startknapp slange
PAST21_0K 4500.00 BOOL  ; FRA NODE3 3100
PAST21_0K_NX 2812.00 BOOL  ; FRA NODE3 3100
PAST21_AVSLUTT 4500.03 BOOL  ; FRA NODE3 3103
PAST21_AVSLUTT_NX 2812.03 BOOL  ; FRA NODE3 3103
PAST21_DM 4502.09 BOOL  ; D_VITAMIN
PAST21_DM_N6 2812.12 BOOL  ; D_VITAMIN
PAST21_DREN_L3_VALG 326.00 BOOL  ; INDIVIDVALG
PAST21_DREN_L4_VALG 326.01 BOOL  ; INDIVIDVALG FRA KOEREGISTER.
PAST21_DREN_TID_S T0536 BOOL  ; X
PAST21_DREN_TID_T 0536 NUMBER
PAST21_DREN_UT 4500.05 BOOL  ; FRA NODE3
PAST21_DREN_UT_NX 2812.04 BOOL  ; FRA NODE3
PAST21_EX 4500.14 BOOL  ; FRA NODE3 3113
PAST21_EX_NX 2812.09 BOOL  ; FRA NODE3 3113
PAST21_FLOETE_UT 4502.03 BOOL  ; FLOETE TIL T24.01
PAST21_FLOETE_V_T2401 4502.02 BOOL  ; FLOETE VED T24.01
PAST21_FLOETE_V_T2401_S T0829 BOOL  ; FLOETE VED T24.01
PAST21_FRA_RUNL_UT 4800.14 BOOL  ; FRA RUNDLOP TIL UYKJOERING
PAST21_HM 4500.08 BOOL  ; FRA NODE3 3108
PAST21_HM_NX 2812.05 BOOL  ; FRA NODE3 3108
PAST21_INN_STARTKOMMANDO 326.15 BOOL
PAST21_INN_TID_S T0526 BOOL  ; X
PAST21_INN_TID_T 0526 NUMBER
PAST21_INN_TMU_TID_S T0726 BOOL  ; INKOBLINGSTID TMU NAAR LINJE IKKE AKTIVERES
PAST21_INN_TMU_TID_T 0726 NUMBER  ; MAX-TID TMU OM IKKE LINJE LEGGES
PAST21_LM 4500.09 BOOL  ; FRA NODE3 3109
PAST21_LM_NX 2812.06 BOOL  ; FRA NODE3 3109
PAST21_MELK 4501.15 BOOL  ; MELK I SYSTEM
PAST21_OKO 4502.10 BOOL
PAST21_OKO_NX 2812.10 BOOL  ; FRA NODE3 3143
PAST21_OMSLAG 4800.07 BOOL
PAST21_OMSLAGSPENN D1420 CHANNEL  ; Z
PAST21_OMSLAGSPENN_OPPSKALER OPPSKALERING
PAST21_PROD 4500.01 BOOL  ; DRIFT PAA PASTEUR21 3101
PAST21_PROD_L3_VALG 326.02 BOOL  ; INDIVIDVALG FRA KOEREGISTER.
PAST21_PROD_L4_VALG 326.03 BOOL  ; INDIVIDVALG
PAST21_PROD_NX 2812.01 BOOL  ; DRIFT PAA PASTEUR21 3101
PAST21_PROD_V2114_S T0831 BOOL  ; FORSINKER RESET AV V2114
PAST21_PROD_V2114_T 0831 NUMBER  ; FORSINKER RESET AV V2114
PAST21_RUNDL 4500.02 BOOL  ; FRA NODE3 3102
PAST21_RUNDL_NX 2812.02 BOOL  ; FRA NODE3 3102
PAST21_SK 4500.10 BOOL  ; FRA NODE3 3110
PAST21_SK_NX 2812.07 BOOL  ; FRA NODE3 3110
PAST21_SOT 4500.12 BOOL  ; FRA NODE3 3111
PAST21_SOT_NX 2812.08 BOOL  ; FRA NODE3 3111
PAST21_SUM_PROD 4801.00 BOOL  ; PROD ELLER DREN ELLER AVSLUTNING
PAST21_TVANG_UT 4500.04 BOOL
PAST21_UHT 4502.11 BOOL  ; ¨
PAST21_UREN 4502.00 BOOL
PAST21_UT 4801.05 BOOL  ; RUNDLOEP AV OG V2144=1
PAST21_UT_NX 2812.11 BOOL  ; RUNDLOEP AV OG V2144=1
PAST21_UT_OK 4801.04 BOOL  ; LINJER FRA  PAST21 TIL TANKER OK
PAST21_VANN 4502.01 BOOL
PAST21_VANN_V_T2401_S T0830 BOOL  ; VANN VED T24.01 I AVSLUTNING
PAST21_VANN_V_T2401_T 0830 NUMBER  ; VANN VED T24.01 I AVSLUTNING
PAST22_0K 4510.00 BOOL  ; FRA NODE3 3200
PAST22_AMPER D2440 WORD  ; PAST 22 MOTORSTROEM. 1000=100,0 AMP
PAST22_AVSLUTT 4510.03 BOOL  ; FRA NODE3 3203
PAST22_DM 4512.09 BOOL  ; D_VITAMIN
PAST22_DM_N6 2827.13 BOOL  ; D_VITAMIN
PAST22_DREN_L3_VALG 327.00 BOOL  ; INDIVIDVALG
PAST22_DREN_L4_VALG 327.01 BOOL  ; INDIVIDVALG FRA KOEREGISTER.
PAST22_DREN_TID_S T0537 BOOL  ; X
PAST22_DREN_TID_T 0537 NUMBER
PAST22_DREN_UT 4510.05 BOOL  ; FRA NODE3 3205
PAST22_EX 4510.14 BOOL  ; FRA NODE3 3213
PAST22_FLOETE_UT 4512.03 BOOL  ; FLOETE TIL T24.01
PAST22_FLOETE_V_T2401 4512.02 BOOL  ; FLOETE VED T24.01
PAST22_FLOETE_V_T2401_S T0833 BOOL  ; FLOETE VED T24.01
PAST22_FLOETE_V_T2401_T 0833 NUMBER  ; FLOETE VED T24.01
PAST22_FRA_RUNL_UT 4810.14 BOOL  ; FRA RUNDLOP TIL UYKJOERING
PAST22_HM 4510.08 BOOL  ; FRA NODE3 3208
PAST22_HM_SIST 4811.08 BOOL  ; HM SISTE PRODUKT
PAST22_INN_STARTKOMMANDO 327.15 BOOL
PAST22_INN_TID_S T0527 BOOL  ; X
PAST22_INN_TID_T 0527 NUMBER
PAST22_INN_TMU_TID_S T0727 BOOL  ; INKOBLINGSTID TMU NAAR LINJE IKKE AKTIVERES
PAST22_INN_TMU_TID_T 0727 NUMBER  ; MAX-TID TMU OM IKKE LINJE LEGGES
PAST22_LM 4510.09 BOOL  ; FRA NODE3 3209
PAST22_LM_SIST 4811.09 BOOL  ; LM SISTE PRODUKT
PAST22_MELK 4511.15 BOOL  ; MELK I SYSTEM
PAST22_MENDE_UHT_OK 4822.03 BOOL
PAST22_OKO 4512.10 BOOL
PAST22_OMSLAG 4810.07 BOOL
PAST22_OMSLAGSPENN D1422 CHANNEL  ; Z
PAST22_OMSLAGSPENN_OPPSKALER OPPSKALERING
PAST22_PROD 4510.01 BOOL  ; FRA NODE3 3201
PAST22_PROD_L3_VALG 327.02 BOOL  ; INDIVIDVALG FRA KOEREGISTER.
PAST22_PROD_L4_VALG 327.03 BOOL  ; INDIVIDVALG
PAST22_PROD_V2214_S T0835 BOOL  ; FORSINKER RESET AV V2214
PAST22_PROD_V2214_T 0835 NUMBER  ; FORSINKER RESET AV V2214
PAST22_RUNDL 4510.02 BOOL  ; FRA NODE3 3202
PAST22_SK 4510.10 BOOL  ; FRA NODE3 3210
PAST22_SK_SIST 4811.10 BOOL  ; SKUMMET SISTE PRODUKT
PAST22_SOT 4510.12 BOOL  ; FRA NODE3 3211
PAST22_SOT_SIST 4811.06 BOOL  ; SOETT PRODUKT SISTE
PAST22_STOPP_ETTER_DREN 4821.02 BOOL  ; ¨
PAST22_SUM_PROD 4811.00 BOOL  ; PROD ELLER DREN ELLER AVSLUTNING
PAST22_SUR 4510.13 BOOL  ; FRA NODE3 3212
PAST22_SUR_SIST 4811.07 BOOL  ; SURT PRODUKT SISTE
PAST22_TVANG_UT 4510.04 BOOL
PAST22_UHT 4512.11 BOOL
PAST22_UREN 4512.00 BOOL
PAST22_UT 4811.05 BOOL  ; RUNDLOEP AV OG V2244=1
PAST22_UT_OK 4811.04 BOOL  ; LINJER FRA  PAST22 TIL TANKER OK
PAST22_VANN 4512.01 BOOL  ; VANN I  SYSTEM
PAST22_VANN_V_T2401_S T0834 BOOL  ; VANN VED T24.01 I AVSLUTNING
PAST22_VANN_V_T2401_T 0834 NUMBER  ; VANN VED T24.01 I AVSLUTNING
PAST22_VIBRASJON D2442 WORD  ; PAST 22_VIBRASJON 2000=20,00mm/S
PAST23_AVSLUTT 4520.03 BOOL  ; FRA NODE3 3103
PAST23_BLK_FLOTE_INN_S T0839 BOOL  ; FORSINKER BUNNSIGNAL BLK
PAST23_BLK_TOM_AVSLUTT 4522.06 BOOL
PAST23_BLK_TOM_FLOTE_INN 4522.04 BOOL  ; ¨
PAST23_BLK_TOM_FLOTE_INN_T 0839 NUMBER  ; FORSINKER BUNNSIGNAL BLK
PAST23_DREN_L3_VALG 328.00 BOOL  ; INDIVIDVALG
PAST23_DREN_L4_VALG 328.01 BOOL  ; INDIVIDVALG FRA KOEREGISTER.
PAST23_DREN_UT 4520.05 BOOL  ; ¨
PAST23_DR_TIL_CONT 4822.02 BOOL
PAST23_FLOTE 4520.11 BOOL
PAST23_FLOTE_INN 4522.05 BOOL
PAST23_FLOTE_INN_S T0840 BOOL  ; FORSINK SINAL FLOETE I BLK
PAST23_FLOTE_I_SYSTEM 4521.15 BOOL
PAST23_FL_INN_T2009_IMP D3880 INT  ; FLOETE  IROER TIL T20.09 NAAR TELLER NAAR FORVALG
PAST23_FL__INNE_GR10 4822.04 BOOL  ; FLOETE I ROER TOL GR.10
PAST23_FL__INNE_T2009 4822.05 BOOL  ; FLOETE IROER TIL T20.09
PAST23_FL__INNE_T2009_N5 2807.03 BOOL  ; FLOETE IROER TIL T20.09
PAST23_FL__INNE_T2009_S T0841 BOOL  ; FLOETE IROER TIL T20.09 UT
PAST23_FL__INNE_T2009_T 0841 NUMBER  ; FLOETE IROER TIL T20.09 UT
PAST23_FRA_RUNDL_TIL_UTKJ 4522.12 BOOL
PAST23_FRA_RUNL_UT 4820.14 BOOL  ; FRA RUNDLOP TIL UYKJOERING
PAST23_INN_STARTKOMMANDO 328.15 BOOL
PAST23_INN_TID_S T0528 BOOL  ; X
PAST23_INN_TID_T 0528 NUMBER
PAST23_INN_TMU_TID_S T0728 BOOL  ; INKOBLINGSTID TMU NAAR LINJE IKKE AKTIVERES
PAST23_INN_TMU_TID_T 0728 NUMBER  ; MAX-TID TMU OM IKKE LINJE LEGGES
PAST23_MELK_SYSTEM 4522.07 BOOL  ; TIL GRAFIKK
PAST23_OK 4520.00 BOOL  ; FRA NODE3 3300
PAST23_OMSLAG 4820.07 BOOL
PAST23_OMSLAGSPENN_OPPSKALER OPPSKALERING
PAST23_PENN_FLOWOMSLAG OPPSKALERING
PAST23_PENN_TRYKKOMSLAG OPPSKALERING
PAST23_PROD 4520.01 BOOL  ; 452001
PAST23_RUNDL 4520.02 BOOL
PAST23_SKR_FLOW_OMSLAG D1436 CHANNEL
PAST23_SKR_OMSLAGSPENN D1424 CHANNEL
PAST23_SKR_TR_OMSLAG D1434 CHANNEL
PAST23_SPERR_FLOTE_TIL_PAST 4522.08 BOOL
PAST23_SUM_PROD 4821.00 BOOL  ; PROD ELLER DREN ELLER AVSLUTNING
PAST23_TIL_CONT 4822.01 BOOL
PAST23_TVANG_UT 4520.04 BOOL
PAST23_VANN_I_SYSTEM 4522.01 BOOL
PAST_COND_VENTE_S T0846 BOOL
PAST_LUT_INN 1338.09 BOOL  ; LUT INN SIGNAL FRA NODE3
PAST_LUT_UT 1338.10 BOOL  ; 133812
PAST_SYRE_INN 1338.11 BOOL  ; SYRE INN SIGNAL FRA NODE3
PAST_SYRE_IUT 1338.12 BOOL  ; SYRE UT SIGNAL FRA NODE3
PEER_N5_06_00 2806.00 BOOL
PEER_N5_06_01 2806.01 BOOL
PEER_N5_06_02 2806.02 BOOL
PEER_N5_06_06 2806.06 BOOL
PEER_N5_06_07 2806.07 BOOL
PEER_N5_06_08 2806.08 BOOL
PEER_N5_06_09 2806.09 BOOL
PEER_N5_06_10 2806.10 BOOL
PEER_N5_06_11 2806.11 BOOL
PEER_N5_06_12 2806.12 BOOL
PEER_N5_06_13 2806.13 BOOL
PGM501_0_STATUS_N5 2810.00 BOOL
PGM501_1_STATUS_N5 2810.01 BOOL
PGM501_2_STATUS_N5 2810.02 BOOL
PGM501_IKKE_FEIL_N5 2810.03 BOOL
PGM501_IND_C03_N5 2828.00 BOOL
PGM501_IND_C05_N5 2828.03 BOOL
PGM501_IND_C06_N5 2828.06 BOOL
PGM501_IND_C07_N5 2828.07 BOOL
PGM501_IND_C08_N5 2828.08 BOOL
PGM501_IND_C32_N5 2828.05 BOOL
PGM501_IND_C50_N5 2828.09 BOOL
PGM501_IND_C52_N5 2828.10 BOOL
PGM501_IND_C53_N5 2828.11 BOOL
PGM501_IND_C54_N5 2828.12 BOOL
PGM501_IND_C77_N5 2828.13 BOOL
PGM501_IND_C78_N5 2828.14 BOOL
PGM501_IND_C79 2828.15 BOOL
PGM501_IND_C83_N5 2828.01 BOOL
PGM501_IND_C84_N5 2828.04 BOOL
PGM501_IND_C86_N5 2828.02 BOOL
PGM501_TMU_N5 2810.04 BOOL
PGM503_0_STATUS 503.01 BOOL  ; XX
PGM503_1_STATUS 503.02 BOOL  ; Z
PGM503_2_STATUS 503.03 BOOL  ; Z
PGM503_DRIFT 503.00 BOOL  ; XX
PGM503_FEIL 503.04 BOOL  ; Z
PGM503_FEILTID 503.05 BOOL  ; Z
PGM503_FEILTID_S T0503 BOOL
PGM503_FEILTID_T 0503 NUMBER
PGM503_INDKON 503.06 BOOL  ; Z
PGM503_IND_C23 1203.00 BOOL  ; VASK PAST21
PGM503_IND_C23_VALG 303.00 BOOL
PGM503_IND_INNE 503.15 BOOL  ; Z
PGM503_KOMMANDO_KOE 303.15 BOOL
PGM503_OFF_IMPULS 503.14 BOOL  ; Z
PGM503_ONIMPULS 503.11 BOOL  ; Z
PGM503_RESET 503.09 BOOL  ; Z
PGM503_START 503.07 BOOL  ; Z
PGM503_STARTIMPULS 503.10 BOOL  ; Z
PGM503_TMU 503.08 BOOL
PGM503_TMU_TID_S T0703 BOOL  ; MAX-TID TMU OM IKKE LINJE LEGGES
PGM503_TMU_TID_T 0703 NUMBER  ; MAX-TID TMU OM IKKE LINJE LEGGES
PGM503_V2104_TID_S T0069 BOOL  ; FRAFALL
PGM503_V2104_TID_T 0069 NUMBER  ; MAX-TID TMU OM IKKE LINJE LEGGES
PGM503_V2204_OPPV 4504.02 BOOL  ; PAST21
PGM504_0_STATUS 504.01 BOOL  ; XX
PGM504_1_STATUS 504.02 BOOL  ; Z
PGM504_2_STATUS 504.03 BOOL  ; Z
PGM504_DRIFT 504.00 BOOL  ; XX
PGM504_FEIL 504.04 BOOL  ; Z
PGM504_FEILTID 504.05 BOOL  ; Z
PGM504_FEILTID_S T0504 BOOL
PGM504_FEILTID_T 0504 NUMBER
PGM504_HC_VASK 4811.13 BOOL  ; VASKE HOLDERCELLE MED EKSTRA FLOW
PGM504_HC_VASK_AVSL 4811.14 BOOL  ; VASKE HOLDERCELLE MED EKSTRA FLOW
PGM504_HC_VASK_TILBM_UTK 4811.15 BOOL  ; VASKE HOLDERCELLE MED EKSTRA FLOW
PGM504_INDKON 504.06 BOOL  ; Z
PGM504_IND_C24 1204.00 BOOL  ; VASK PAST22
PGM504_IND_C24_VALG 304.00 BOOL
PGM504_IND_INNE 504.15 BOOL  ; Z
PGM504_KOMMANDO_KOE 304.15 BOOL
PGM504_OFF_IMPULS 504.14 BOOL  ; Z
PGM504_ONIMPULS 504.11 BOOL  ; Z
PGM504_RESET 504.09 BOOL  ; Z
PGM504_START 504.07 BOOL  ; Z
PGM504_STARTIMPULS 504.10 BOOL  ; Z
PGM504_TMU 504.08 BOOL
PGM504_TMU_TID_S T0704 BOOL  ; MAX-TID TMU OM IKKE LINJE LEGGES
PGM504_TMU_TID_T 0704 NUMBER  ; MAX-TID TMU OM IKKE LINJE LEGGES
PGM504_V2204_OPPV 4514.02 BOOL  ; PAST22
PGM504_V2211_12_VEKSL_S T0071 BOOL  ; FORSINKELSE VED STILLINGSENDRING
PGM504_V2211_12_VEKSL_T 0071 NUMBER  ; FORSINKELSE VED STILLINGSENDRING
PGM505_0_STATUS 505.01 BOOL  ; XX
PGM505_0_STATUS_N5 2823.01 BOOL
PGM505_1_STATUS 505.02 BOOL  ; Z
PGM505_1_STATUS_N5 2823.02 BOOL
PGM505_2_STATUS 505.03 BOOL
PGM505_2_STATUS_N5 2823.03 BOOL
PGM505_DRIFT 505.00 BOOL  ; XX
PGM505_FEIL 505.04 BOOL  ; Z
PGM505_FEILTID 505.05 BOOL  ; Z
PGM505_IKKE_FEIL_N5 2823.05 BOOL
PGM505_INDIVID_N5 2823.00 BOOL
PGM505_INDKON 505.06 BOOL  ; Z
PGM505_IND_C25_VALG 305.00 BOOL
PGM505_IND_INNE 505.15 BOOL  ; Z
PGM505_KOMMANDO_KOE 305.15 BOOL
PGM505_OFF_IMPULS 505.14 BOOL  ; Z
PGM505_ONIMPULS 505.11 BOOL  ; Z
PGM505_RESET 505.09 BOOL  ; Z
PGM505_START 505.07 BOOL  ; Z
PGM505_STARTIMPULS 505.10 BOOL  ; Z
PGM505_TID_S T0505 BOOL  ; X
PGM505_TID_T 0505 NUMBER  ; X
PGM505_TMU 505.08 BOOL
PGM505_TMU_N5 2823.04 BOOL
PGM505_TMU_TID_S T0705 BOOL  ; MAX-TID TMU OM IKKE LINJE LEGGES
PGM505_TMU_TID_T 0705 NUMBER  ; MAX-TID TMU OM IKKE LINJE LEGGES
PGM510_0_STAT 510.01 BOOL
PGM510_0_STATUS_N5 2801.02 BOOL
PGM510_1_STAT 510.02 BOOL
PGM510_1_STATUS_N5 2801.03 BOOL
PGM510_2_STAT 510.03 BOOL
PGM510_2_STATUS_N5 2801.04 BOOL
PGM510_DRIFT 510.00 BOOL
PGM510_DRIFT_N5 2801.01 BOOL
PGM510_FEIL 510.04 BOOL
PGM510_FEILTID 510.05 BOOL
PGM510_FEILTID_S T0510 BOOL
PGM510_FEILTID_T 0510 NUMBER
PGM510_IKKE_FEIL_N5 2801.05 BOOL
PGM510_IND_C26 1210.03 BOOL  ; T20.02
PGM510_IND_C26_N5 2815.03 BOOL  ; T20.02
PGM510_IND_C27 1210.04 BOOL  ; T20.33 (03)
PGM510_IND_C27_N5 2815.04 BOOL  ; T20.33 (03)
PGM510_IND_C28 1210.05 BOOL  ; T20.34 (04)
PGM510_IND_C28_N5 2815.05 BOOL  ; T20.34 (04)
PGM510_IND_C29 1210.06 BOOL  ; T20.35 (05)
PGM510_IND_C29_N5 2815.06 BOOL  ; T20.35 (05)
PGM510_IND_C80 1210.02 BOOL  ; RV T20.28-T20.29
PGM510_IND_C80_N5 2815.02 BOOL  ; RV T20.28-T20.29
PGM510_IND_C87 1210.07 BOOL
PGM510_IND_C87_N5 2815.07 BOOL
PGM510_IND_C88 1210.08 BOOL  ; T20.30 SCANIMA
PGM510_IND_C88_N5 2815.08 BOOL  ; T20.30 SCANIMA
PGM510_IND_C89 1210.09 BOOL
PGM510_IND_C89_N5 2815.09 BOOL
PGM510_IND_C90 1210.00 BOOL  ; T20.28
PGM510_IND_C90_N5 2815.00 BOOL  ; T20.28
PGM510_IND_C91 1210.01 BOOL  ; T20.29
PGM510_IND_C91_N5 2815.01 BOOL  ; T20.29
PGM510_IND_C92 1210.10 BOOL  ; RV STERIL
PGM510_IND_C92_N5 2815.10 BOOL  ; RV STERIL
PGM510_IND_INNE_HJ1 910.10 BOOL
PGM510_IND_INNE_HJ2 910.11 BOOL
PGM510_START 510.07 BOOL
PGM510_STOPP 510.09 BOOL
PGM510_STOPP_N5 2801.00 BOOL
PGM510_TMU 510.08 BOOL
PGM511_0_STAT 511.01 BOOL
PGM511_0_STAT_N5 2801.10 BOOL
PGM511_1_STAT 511.02 BOOL
PGM511_1_STAT_N5 2801.11 BOOL
PGM511_2_STAT 511.03 BOOL
PGM511_2_STAT_N5 2801.12 BOOL
PGM511_C45_LINJETOEM 2955.09 BOOL
PGM511_DRIFT 511.00 BOOL
PGM511_DRIFT_N5 2801.09 BOOL
PGM511_FEIL 511.04 BOOL
PGM511_FEILTID 511.05 BOOL
PGM511_FEILTID_S T0011 BOOL
PGM511_FEILTID_T 011 NUMBER
PGM511_HJ1 900.12 BOOL
PGM511_HJ2 900.13 BOOL
PGM511_IKKE_FEIL_N5 2801.13 BOOL
PGM511_IND_C39 1211.00 BOOL  ; T20.11
PGM511_IND_C39_N5 2816.00 BOOL  ; T20.11
PGM511_IND_C40 1211.01 BOOL  ; T20.12
PGM511_IND_C40_N5 2816.01 BOOL  ; T20.12
PGM511_IND_C41 1211.02 BOOL  ; T20.14
PGM511_IND_C41_N5 2816.02 BOOL  ; T20.14
PGM511_IND_C42 1211.03 BOOL  ; T20.13
PGM511_IND_C42_N5 2816.03 BOOL  ; T20.13
PGM511_IND_C43 1211.04 BOOL  ; T20.16
PGM511_IND_C43_N5 2816.04 BOOL  ; T20.16
PGM511_IND_C44 1211.05 BOOL  ; T20.15
PGM511_IND_C44_N5 2816.05 BOOL  ; T20.15
PGM511_IND_C45 1211.06 BOOL  ; RV
PGM511_IND_C45_N5 2816.06 BOOL  ; RV
PGM511_IND_C47 1211.07 BOOL  ; T20.19
PGM511_IND_C47_N5 2816.07 BOOL  ; T20.19
PGM511_IND_C48 1211.08 BOOL  ; T20.09
PGM511_IND_C48_N5 2816.08 BOOL  ; T20.09
PGM511_IND_C49 1211.09 BOOL  ; RV
PGM511_IND_C49_N5 2816.09 BOOL  ; RV
PGM511_IND_C57 1211.10 BOOL  ; T20.18
PGM511_IND_C57_N5 2816.10 BOOL  ; T20.18
PGM511_IND_C58 1211.11 BOOL  ; T20.17
PGM511_IND_C58_N5 2816.11 BOOL  ; T20.17
PGM511_IND_C93 1211.12 BOOL  ; T20.36
PGM511_IND_C93_N5 2816.12 BOOL  ; T20.36
PGM511_IND_C94 1211.13 BOOL  ; T20.37
PGM511_IND_C94_N5 2816.13 BOOL  ; T20.37
PGM511_IND_INNE_HJ1 910.12 BOOL
PGM511_IND_INNE_HJ2 910.13 BOOL
PGM511_START 511.07 BOOL
PGM511_STOPP 511.09 BOOL
PGM511_STOPP_N5 2801.08 BOOL
PGM511_TMU 511.08 BOOL
PGM511_TMU_N5 2931.10 BOOL
PGM512_FEILTID_S T0012 BOOL
PGM512_FEILTID_T 012 NUMBER
PGM512_IND_C55 1212.00 BOOL  ; TV-STERIL
PGM512_IND_C55_N5 2817.00 BOOL  ; TV_STERILOMRAADET
PGM512_IND_C56 1212.01 BOOL  ; RV-STERIL
PGM512_IND_C56_N5 2817.01 BOOL  ; RV_STERILOMRAADET
PGM512_IND_INNE_HJ1 910.14 BOOL
PGM512_IND_INNE_HJ2 910.15 BOOL
PGM514_C60_VALG_VST60_K1 314.00 BOOL  ; Z
PGM514_C61_VALG_VST60_K1 314.01 BOOL  ; Z
PGM514_C62_VALG_VST60_K1 314.02 BOOL  ; Z
PGM514_C63_VALG_VST60_K1 314.03 BOOL  ; Z
PGM514_C64_VALG_VST60_K1 314.04 BOOL  ; Z
PGM514_C65_VALG_VST60_K1 314.05 BOOL  ; Z
PGM514_C66_VALG_VST60_K1 314.06 BOOL  ; Z
PGM514_C67_VALG_VST60_K1 314.07 BOOL  ; Z
PGM514_C68_VALG_VST60_K1 314.08 BOOL
PGM514_C69_VALG_VST60_K1 314.09 BOOL
PGM514_C70_VALG_VST60_K1 314.10 BOOL
PGM514_C71_VALG_VST60_K1 314.11 BOOL
PGM514_C72_VALG_VST60_K1 314.12 BOOL
PGM514_C73_VALG_VST60_K1 314.13 BOOL
PGM514_C74_VALG_VST60_K1 314.14 BOOL
PGM514_C75_VALG_VST60_K1 314.15 BOOL
PGM514_KOMMANDO_KOE 414.00 BOOL
PGM515_0_STATUS 515.01 BOOL
PGM515_0_STATUS_N5 2809.02 BOOL
PGM515_1_STATUS 515.02 BOOL
PGM515_1_STATUS_N5 2809.03 BOOL
PGM515_2_STATUS 515.03 BOOL
PGM515_2_STATUS_N5 2809.04 BOOL
PGM515_DRIFT 515.00 BOOL
PGM515_DRIFT_N5 2809.01 BOOL
PGM515_FEIL 515.04 BOOL
PGM515_FEILTID 515.05 BOOL
PGM515_IKKE_FEIL_N5 2809.05 BOOL
PGM515_IND_C16 1215.00 BOOL
PGM515_IND_C17 1215.01 BOOL
PGM515_IND_C18 1215.02 BOOL
PGM515_IND_C19 1215.03 BOOL
PGM515_IND_C20 1215.04 BOOL
PGM515_IND_C21 1215.07 BOOL
PGM515_IND_C22 1215.05 BOOL
PGM515_IND_C46 1215.08 BOOL
PGM515_IND_C76 1215.06 BOOL
PGM515_START 515.07 BOOL
PGM515_STOPP 515.09 BOOL
PGM515_STOPP_N5 2809.00 BOOL
PGM515_STOPP_S T0823 BOOL
PGM515_STOPP_T 0823 NUMBER
PGM515_TID_S T0515 BOOL  ; X
PGM515_TID_T 0515 NUMBER  ; X
PGM515_TIL_TGR08_IND_N5 2809.00 BOOL
PGM528_IND_L3 1228.00 BOOL
PGM528_IND_L4 1228.01 BOOL
PGM529_0_STATUS 529.01 BOOL  ; Z
PGM529_1_STATUS 529.02 BOOL  ; Z
PGM529_2_STATUS 529.03 BOOL  ; Z
PGM529_DRIFT 529.00 BOOL  ; XX
PGM529_FEIL 529.04 BOOL  ; Z
PGM529_FEILTID 529.05 BOOL  ; Z
PGM529_FEILTID_S T0529 BOOL
PGM529_INDKON 529.06 BOOL  ; Z
PGM529_IND_CONT 1229.01 BOOL  ; FRA CONTEINER
PGM529_IND_CONT_VALG 329.01 BOOL  ; FRA CONTEINER
PGM529_IND_INNE 529.15 BOOL  ; Z
PGM529_IND_T24 1229.00 BOOL
PGM529_IND_T24_VALG 329.00 BOOL
PGM529_KOMMANDO_KOE 329.15 BOOL
PGM529_OFF_IMPULS 529.14 BOOL  ; Z
PGM529_ONIMPULS 529.11 BOOL  ; Z
PGM529_RESET 529.09 BOOL  ; Z
PGM529_START 529.07 BOOL  ; Z
PGM529_STARTIMPULS 529.10 BOOL  ; Z
PGM529_TMU 529.08 BOOL
PGM529_TMU_TID_S T0729 BOOL  ; MAX-TID TMU OM IKKE LINJE LEGGES
PGM530_0_STATUS 530.01 BOOL  ; PAST21 TIL UHT
PGM530_0_STATUS_N5 2830.02 BOOL  ; PAST21 TIL UHT
PGM530_1_STATUS 530.02 BOOL  ; PAST21 TIL UHT
PGM530_1_STATUS_N5 2830.03 BOOL  ; PAST21 TIL UHT
PGM530_2_STAT 530.03 BOOL  ; PAST21 TIL UHT
PGM530_2_STAT_N5 2830.04 BOOL  ; PAST21 TIL UHT
PGM530_DIREKTE_IND 1230.04 BOOL
PGM530_DRIFT 530.00 BOOL  ; PAST21 TIL UHT
PGM530_DRIFT_N5 2830.01 BOOL  ; PAST21 TIL UHT
PGM530_FEIL 530.04 BOOL  ; PAST21 TIL UHT
PGM530_FEILTID 530.05 BOOL  ; PAST21 TIL UHT
PGM530_FEILTID_S T0530 BOOL
PGM530_FEILTID_T 0530 NUMBER
PGM530_IKKE_FEIL_N5 2830.05 BOOL  ; PAST21 TIL UHT
PGM530_START 530.07 BOOL  ; PAST21 TIL UHT
PGM530_STOPP 530.09 BOOL  ; PAST21 TIL UHT
PGM530_STOPP_N5 2830.00 BOOL  ; PAST21 TIL UHT
PGM530_T2009_IND 1230.00 BOOL
PGM530_T2033_IND 1230.01 BOOL
PGM530_T2034_IND 1230.02 BOOL
PGM530_T2035_IND 1230.03 BOOL
PGM531_0_STATUS 531.01 BOOL  ; PAST22 TIL UHT
PGM531_0_STATUS_N5 2830.10 BOOL  ; PAST22 TIL UHT
PGM531_1_STATUS 531.02 BOOL  ; PAST22 TIL UHT
PGM531_1_STATUS_N5 2830.11 BOOL  ; PAST22 TIL UHT
PGM531_2_STAT 531.03 BOOL  ; PAST22 TIL UHT
PGM531_2_STAT_N5 2830.12 BOOL  ; PAST22 TIL UHT
PGM531_DIREKTE_IND 1231.03 BOOL
PGM531_DRIFT 531.00 BOOL  ; PAST22 TIL UHT
PGM531_DRIFT_N5 2830.09 BOOL  ; PAST22 TIL UHT
PGM531_FEIL 531.04 BOOL  ; PAST22 TIL UHT
PGM531_FEILTID 531.05 BOOL  ; PAST22 TIL UHT
PGM531_FEILTID_S T0531 BOOL
PGM531_FEILTID_T 0531 NUMBER
PGM531_IKKE_FEIL_N5 2830.13 BOOL  ; PAST22 TIL UHT
PGM531_START 531.07 BOOL  ; PAST22 TIL UHT
PGM531_STOPP 531.09 BOOL  ; PAST22 TIL UHT
PGM531_STOPP_N5 2830.08 BOOL  ; PAST22 TIL UHT
PGM531_T2033_IND 1231.00 BOOL
PGM531_T2034_IND 1231.01 BOOL
PGM531_T2035_IND 1231.02 BOOL
PGM532_0_STATUS 532.01 BOOL  ; PAST23 TIL UHT
PGM532_0_STATUS_N5 2831.02 BOOL  ; PAST23 TIL UHT
PGM532_1_STATUS 532.02 BOOL  ; PAST23 TIL UHT
PGM532_1_STATUS_N5 2831.03 BOOL  ; PAST23 TIL UHT
PGM532_2_STAT 532.03 BOOL  ; PAST23 TIL UHT
PGM532_2_STAT_N5 2831.04 BOOL  ; PAST23 TIL UHT
PGM532_DIREKTE_IND 1232.03 BOOL
PGM532_DRIFT 532.00 BOOL  ; PAST23 TIL UHT
PGM532_DRIFT_N5 2831.01 BOOL  ; PAST23 TIL UHT
PGM532_FEIL 532.04 BOOL  ; PAST23 TIL UHT
PGM532_FEILTID 532.05 BOOL  ; PAST23 TIL UHT
PGM532_FEILTID_S T0532 BOOL
PGM532_FEILTID_T 0532 NUMBER
PGM532_IKKE_FEIL_N5 2831.05 BOOL  ; PAST23 TIL UHT
PGM532_START 532.07 BOOL  ; PAST23 TIL UHT
PGM532_STOPP 532.09 BOOL  ; PAST23 TIL UHT
PGM532_STOPP_N5 2831.00 BOOL  ; PAST23 TIL UHT
PGM532_T2033_IND 1232.00 BOOL
PGM532_T2034_IND 1232.01 BOOL
PGM532_T2035_IND 1232.02 BOOL
PGM535_FEILTID_S T0535 BOOL
PGM535_FEILTID_T 0535 NUMBER
PGM535_START 537.07 BOOL
PGM539_0_STATUS 539.01 BOOL
PGM539_1_STATUS 539.02 BOOL
PGM539_2_STATUS 539.03 BOOL
PGM539_DRIFT 539.00 BOOL
PGM539_FEIL 539.04 BOOL
PGM539_FEILTID 539.05 BOOL
PGM539_FEILTID_S T0539 BOOL
PGM539_FEILTID_T 0539 NUMBER
PGM539_IND_INNE_HJ1 910.00 BOOL
PGM539_IND_INNE_HJ2 910.01 BOOL
PGM539_IND_TIL_T2011 1239.00 BOOL  ; TIL
PGM539_IND_TIL_T2012 1239.01 BOOL
PGM539_IND_TIL_T2013 1239.02 BOOL
PGM539_IND_TIL_T2014 1239.03 BOOL
PGM539_IND_TIL_T2015 1239.04 BOOL
PGM539_IND_TIL_T2016 1239.05 BOOL
PGM539_IND_TIL_T2017 1239.06 BOOL
PGM539_IND_TIL_T2018 1239.07 BOOL
PGM539_IND_TIL_T2019 1239.08 BOOL
PGM539_IND_TIL_T2036 1239.09 BOOL
PGM539_IND_TIL_T2037 1239.10 BOOL
PGM539_START 539.07 BOOL
PGM539_STOPP 539.09 BOOL
PGM540_IND_T2011_P2031_N5 2811.00 BOOL
PGM540_IND_T2012_P2031_N5 2811.01 BOOL
PGM540_IND_T2013_P2031_N5 2811.02 BOOL
PGM540_IND_T2014_P2031_N5 2811.03 BOOL
PGM540_IND_T2015_P2031_N5 2811.04 BOOL
PGM540_IND_T2016_P2031_N5 2811.05 BOOL
PGM540_IND_T2017_P2031_N5 2811.06 BOOL
PGM540_IND_T2018_P2031_N5 2811.07 BOOL
PGM540_IND_T2019_P2031_N5 2811.08 BOOL
PGM540_IND_T2036_P2031_N5 2811.09 BOOL
PGM540_IND_T2037_P2031_N5 2811.10 BOOL
PGM544_0_STATUS 544.01 BOOL  ; BIL TI OEKOMELKTANK T27.01
PGM544_1_STATUS 544.02 BOOL  ; BIL TI OEKOMELKTANK T27.01
PGM544_2_STATUS 544.03 BOOL  ; BIL TI OEKOMELKTANK T27.01
PGM544_DRIFT 544.00 BOOL  ; BIL TI OEKOMELKTANK T27.01
PGM544_FEIL 544.04 BOOL  ; BIL TI OEKOMELKTANK T27.01
PGM544_FEILTID 544.05 BOOL  ; BIL TI OEKOMELKTANK T27.01
PGM544_FEILTID_S T0544 BOOL
PGM544_INDIVID_INNE 544.15 BOOL  ; BIL TI OEKOMELKTANK T27.01
PGM544_INDKON 544.06 BOOL  ; BIL TI OEKOMELKTANK T27.01
PGM544_IND_00 1244.00 BOOL  ; BIL TIL T2701
PGM544_IND_VALG 344.00 BOOL  ; INDIVIDVALG
PGM544_OFF_IMP 544.14 BOOL  ; BIL TI OEKOMELKTANK T27.01
PGM544_ONIMPULS 544.11 BOOL  ; BIL TI OEKOMELKTANK T27.01
PGM544_START 544.07 BOOL  ; BIL TI OEKOMELKTANK T27.01
PGM544_STARTKOMMANDO 344.15 BOOL
PGM544_STOPP 544.09 BOOL  ; BIL TI OEKOMELKTANK T27.01
PGM544_TMU_TID_S T0744 BOOL  ; MAX-TID TMU OM IKKE LINJE LEGGES
PGM544_TMU_USIKRET 544.08 BOOL  ; BIL TI OEKOMELKTANK T27.01
PGM546_0_STATUS 546.01 BOOL  ; PAST23 TIL T2009
PGM546_0_STATUS_N5 2831.10 BOOL
PGM546_1_STATUS 546.02 BOOL  ; PAST23 TIL T2009
PGM546_1_STATUS_N5 2831.11 BOOL
PGM546_2_STAT 546.03 BOOL  ; PAST23 TIL T2009
PGM546_2_STAT_N5 2831.12 BOOL
